LIN {X 9.053,Y 108.159,Z 56.000,A 180.000,B 0.000,C 180.000} C_DIS
LIN {X 9.120,Y 108.308,Z 56.000,A 180.000,B 0.000,C 180.000} C_DIS
LIN {X 9.797,Y 109.768,Z 56.000,A 180.000,B 0.000,C 180.000} C_DIS
LIN {X 9.836,Y 109.849,Z 56.000,A 180.000,B 0.000,C 180.000} C_DIS
LIN {X 10.551,Y 111.303,Z 56.000,A 180.000,B 0.000,C 180.000} C_DIS
LIN {X 10.587,Y 111.377,Z 56.000,A 180.000,B 0.000,C 180.000} C_DIS
LIN {X 10.680,Y 111.556,Z 56.000,A 180.000,B 0.000,C 180.000} C_DIS
LIN {X 11.332,Y 112.807,Z 56.000,A 180.000,B 0.000,C 180.000} C_DIS
LIN {X 11.426,Y 112.986,Z 56.000,A 180.000,B 0.000,C 180.000} C_DIS
LIN {X 12.215,Y 114.416,Z 56.000,A 180.000,B 0.000,C 180.000} C_DIS
LIN {X 12.317,Y 114.595,Z 56.000,A 180.000,B 0.000,C 180.000} C_DIS
LIN {X 13.053,Y 115.859,Z 56.000,A 180.000,B 0.000,C 180.000} C_DIS
LIN {X 13.151,Y 116.025,Z 56.000,A 180.000,B 0.000,C 180.000} C_DIS
LIN {X 13.232,Y 116.158,Z 56.000,A 180.000,B 0.000,C 180.000} C_DIS
LIN {X 14.029,Y 117.455,Z 56.000,A 180.000,B 0.000,C 180.000} C_DIS
LIN {X 14.126,Y 117.607,Z 56.000,A 180.000,B 0.000,C 180.000} C_DIS
LIN {X 14.953,Y 118.885,Z 56.000,A 180.000,B 0.000,C 180.000} C_DIS
LIN {X 15.020,Y 118.988,Z 56.000,A 180.000,B 0.000,C 180.000} C_DIS
LIN {X 15.072,Y 119.064,Z 56.000,A 180.000,B 0.000,C 180.000} C_DIS
LIN {X 15.924,Y 120.315,Z 56.000,A 180.000,B 0.000,C 180.000} C_DIS
LIN {X 16.047,Y 120.494,Z 56.000,A 180.000,B 0.000,C 180.000} C_DIS
LIN {X 16.986,Y 121.806,Z 56.000,A 180.000,B 0.000,C 180.000} C_DIS
LIN {X 17.073,Y 121.924,Z 56.000,A 180.000,B 0.000,C 180.000} C_DIS
LIN {X 18.059,Y 123.235,Z 56.000,A 180.000,B 0.000,C 180.000} C_DIS
LIN {X 18.152,Y 123.354,Z 56.000,A 180.000,B 0.000,C 180.000} C_DIS
LIN {X 19.139,Y 124.606,Z 56.000,A 180.000,B 0.000,C 180.000} C_DIS
LIN {X 19.286,Y 124.785,Z 56.000,A 180.000,B 0.000,C 180.000} C_DIS
LIN {X 20.204,Y 125.894,Z 56.000,A 180.000,B 0.000,C 180.000} C_DIS
LIN {X 20.323,Y 126.036,Z 56.000,A 180.000,B 0.000,C 180.000} C_DIS
LIN {X 21.410,Y 127.287,Z 56.000,A 180.000,B 0.000,C 180.000} C_DIS
LIN {X 21.456,Y 127.340,Z 56.000,A 180.000,B 0.000,C 180.000} C_DIS
LIN {X 21.570,Y 127.466,Z 56.000,A 180.000,B 0.000,C 180.000} C_DIS
LIN {X 22.547,Y 128.539,Z 56.000,A 180.000,B 0.000,C 180.000} C_DIS
LIN {X 22.707,Y 128.711,Z 56.000,A 180.000,B 0.000,C 180.000} C_DIS
LIN {X 23.780,Y 129.835,Z 56.000,A 180.000,B 0.000,C 180.000} C_DIS
LIN {X 23.910,Y 129.969,Z 56.000,A 180.000,B 0.000,C 180.000} C_DIS
LIN {X 25.031,Y 131.090,Z 56.000,A 180.000,B 0.000,C 180.000} C_DIS
LIN {X 25.165,Y 131.220,Z 56.000,A 180.000,B 0.000,C 180.000} C_DIS
LIN {X 26.289,Y 132.293,Z 56.000,A 180.000,B 0.000,C 180.000} C_DIS
LIN {X 26.461,Y 132.453,Z 56.000,A 180.000,B 0.000,C 180.000} C_DIS
LIN {X 27.534,Y 133.430,Z 56.000,A 180.000,B 0.000,C 180.000} C_DIS
LIN {X 27.660,Y 133.544,Z 56.000,A 180.000,B 0.000,C 180.000} C_DIS
LIN {X 27.713,Y 133.590,Z 56.000,A 180.000,B 0.000,C 180.000} C_DIS
LIN {X 28.964,Y 134.677,Z 56.000,A 180.000,B 0.000,C 180.000} C_DIS
LIN {X 29.106,Y 134.796,Z 56.000,A 180.000,B 0.000,C 180.000} C_DIS
LIN {X 30.215,Y 135.714,Z 56.000,A 180.000,B 0.000,C 180.000} C_DIS
LIN {X 30.394,Y 135.861,Z 56.000,A 180.000,B 0.000,C 180.000} C_DIS
LIN {X 31.646,Y 136.848,Z 56.000,A 180.000,B 0.000,C 180.000} C_DIS
LIN {X 31.765,Y 136.941,Z 56.000,A 180.000,B 0.000,C 180.000} C_DIS
LIN {X 33.076,Y 137.927,Z 56.000,A 180.000,B 0.000,C 180.000} C_DIS
LIN {X 33.194,Y 138.014,Z 56.000,A 180.000,B 0.000,C 180.000} C_DIS
LIN {X 34.506,Y 138.953,Z 56.000,A 180.000,B 0.000,C 180.000} C_DIS
LIN {X 34.685,Y 139.076,Z 56.000,A 180.000,B 0.000,C 180.000} C_DIS
LIN {X 35.936,Y 139.928,Z 56.000,A 180.000,B 0.000,C 180.000} C_DIS
LIN {X 36.012,Y 139.980,Z 56.000,A 180.000,B 0.000,C 180.000} C_DIS
LIN {X 36.115,Y 140.047,Z 56.000,A 180.000,B 0.000,C 180.000} C_DIS
LIN {X 37.393,Y 140.874,Z 56.000,A 180.000,B 0.000,C 180.000} C_DIS
LIN {X 37.545,Y 140.971,Z 56.000,A 180.000,B 0.000,C 180.000} C_DIS
LIN {X 38.842,Y 141.768,Z 56.000,A 180.000,B 0.000,C 180.000} C_DIS
LIN {X 38.975,Y 141.849,Z 56.000,A 180.000,B 0.000,C 180.000} C_DIS
LIN {X 39.141,Y 141.947,Z 56.000,A 180.000,B 0.000,C 180.000} C_DIS
LIN {X 40.405,Y 142.683,Z 56.000,A 180.000,B 0.000,C 180.000} C_DIS
LIN {X 40.584,Y 142.785,Z 56.000,A 180.000,B 0.000,C 180.000} C_DIS
LIN {X 42.014,Y 143.574,Z 56.000,A 180.000,B 0.000,C 180.000} C_DIS
LIN {X 42.193,Y 143.668,Z 56.000,A 180.000,B 0.000,C 180.000} C_DIS
LIN {X 43.444,Y 144.320,Z 56.000,A 180.000,B 0.000,C 180.000} C_DIS
LIN {X 43.623,Y 144.413,Z 56.000,A 180.000,B 0.000,C 180.000} C_DIS
LIN {X 43.697,Y 144.449,Z 56.000,A 180.000,B 0.000,C 180.000} C_DIS
LIN {X 45.151,Y 145.164,Z 56.000,A 180.000,B 0.000,C 180.000} C_DIS
LIN {X 45.232,Y 145.203,Z 56.000,A 180.000,B 0.000,C 180.000} C_DIS
LIN {X 46.692,Y 145.880,Z 56.000,A 180.000,B 0.000,C 180.000} C_DIS
LIN {X 46.841,Y 145.947,Z 56.000,A 180.000,B 0.000,C 180.000} C_DIS
LIN {X 48.331,Y 146.595,Z 56.000,A 180.000,B 0.000,C 180.000} C_DIS
LIN {X 48.450,Y 146.645,Z 56.000,A 180.000,B 0.000,C 180.000} C_DIS
LIN {X 49.880,Y 147.227,Z 56.000,A 180.000,B 0.000,C 180.000} C_DIS
LIN {X 50.059,Y 147.299,Z 56.000,A 180.000,B 0.000,C 180.000} C_DIS
LIN {X 51.496,Y 147.846,Z 56.000,A 180.000,B 0.000,C 180.000} C_DIS
LIN {X 51.668,Y 147.911,Z 56.000,A 180.000,B 0.000,C 180.000} C_DIS
LIN {X 51.847,Y 147.974,Z 56.000,A 180.000,B 0.000,C 180.000} C_DIS
LIN {X 52.272,Y 148.125,Z 56.000,A 180.000,B 0.000,C 180.000} C_DIS
; Link Move Starts
LIN {X 52.569,Y 148.230,Z 56.000,A 180.000,B 0.000,C 180.000} C_DIS
LIN {X 52.866,Y 148.335,Z 55.999,A 180.000,B 0.000,C 180.000} C_DIS
LIN {X 53.163,Y 148.440,Z 55.998,A 180.000,B 0.000,C 180.000} C_DIS
LIN {X 53.461,Y 148.542,Z 55.996,A 180.000,B 0.000,C 180.000} C_DIS
LIN {X 53.761,Y 148.640,Z 55.994,A 180.000,B 0.000,C 180.000} C_DIS
LIN {X 54.060,Y 148.738,Z 55.991,A 180.000,B 0.000,C 180.000} C_DIS
LIN {X 54.359,Y 148.836,Z 55.988,A 180.000,B 0.000,C 180.000} C_DIS
LIN {X 54.659,Y 148.934,Z 55.985,A 180.000,B 0.000,C 180.000} C_DIS
LIN {X 54.958,Y 149.032,Z 55.981,A 180.000,B 0.000,C 180.000} C_DIS
LIN {X 55.260,Y 149.124,Z 55.977,A 180.000,B 0.000,C 180.000} C_DIS
LIN {X 55.561,Y 149.215,Z 55.972,A 180.000,B 0.000,C 180.000} C_DIS
LIN {X 55.712,Y 149.260,Z 55.969,A 180.000,B 0.000,C 180.000} C_DIS
LIN {X 55.863,Y 149.306,Z 55.967,A 180.000,B 0.000,C 180.000} C_DIS
LIN {X 56.013,Y 149.351,Z 55.964,A 180.000,B 0.000,C 180.000} C_DIS
LIN {X 56.164,Y 149.397,Z 55.961,A 180.000,B 0.000,C 180.000} C_DIS
LIN {X 56.315,Y 149.442,Z 55.959,A 180.000,B 0.000,C 180.000} C_DIS
LIN {X 56.466,Y 149.488,Z 55.956,A 180.000,B 0.000,C 180.000} C_DIS
LIN {X 56.617,Y 149.533,Z 55.952,A 180.000,B 0.000,C 180.000} C_DIS
LIN {X 56.768,Y 149.577,Z 55.949,A 180.000,B 0.000,C 180.000} C_DIS
LIN {X 56.920,Y 149.619,Z 55.946,A 180.000,B 0.000,C 180.000} C_DIS
LIN {X 57.072,Y 149.661,Z 55.943,A 180.000,B 0.000,C 180.000} C_DIS
LIN {X 57.223,Y 149.703,Z 55.939,A 180.000,B 0.000,C 180.000} C_DIS
LIN {X 57.375,Y 149.745,Z 55.936,A 180.000,B 0.000,C 180.000} C_DIS
LIN {X 57.527,Y 149.786,Z 55.932,A 180.000,B 0.000,C 180.000} C_DIS
LIN {X 57.679,Y 149.828,Z 55.928,A 180.000,B 0.000,C 180.000} C_DIS
LIN {X 57.831,Y 149.870,Z 55.925,A 180.000,B 0.000,C 180.000} C_DIS
LIN {X 57.982,Y 149.912,Z 55.921,A 180.000,B 0.000,C 180.000} C_DIS
LIN {X 58.134,Y 149.954,Z 55.917,A 180.000,B 0.000,C 180.000} C_DIS
LIN {X 58.286,Y 149.996,Z 55.913,A 180.000,B 0.000,C 180.000} C_DIS
LIN {X 58.438,Y 150.037,Z 55.909,A 180.000,B 0.000,C 180.000} C_DIS
LIN {X 58.591,Y 150.075,Z 55.905,A 180.000,B 0.000,C 180.000} C_DIS
LIN {X 58.744,Y 150.113,Z 55.900,A 180.000,B 0.000,C 180.000} C_DIS
LIN {X 58.897,Y 150.152,Z 55.896,A 180.000,B 0.000,C 180.000} C_DIS
LIN {X 59.049,Y 150.190,Z 55.892,A 180.000,B 0.000,C 180.000} C_DIS
LIN {X 59.202,Y 150.229,Z 55.887,A 180.000,B 0.000,C 180.000} C_DIS
LIN {X 59.355,Y 150.267,Z 55.883,A 180.000,B 0.000,C 180.000} C_DIS
LIN {X 59.508,Y 150.305,Z 55.878,A 180.000,B 0.000,C 180.000} C_DIS
LIN {X 59.660,Y 150.344,Z 55.873,A 180.000,B 0.000,C 180.000} C_DIS
LIN {X 59.813,Y 150.382,Z 55.869,A 180.000,B 0.000,C 180.000} C_DIS
LIN {X 59.966,Y 150.420,Z 55.864,A 180.000,B 0.000,C 180.000} C_DIS
LIN {X 60.119,Y 150.458,Z 55.859,A 180.000,B 0.000,C 180.000} C_DIS
LIN {X 60.272,Y 150.493,Z 55.854,A 180.000,B 0.000,C 180.000} C_DIS
LIN {X 60.349,Y 150.510,Z 55.851,A 180.000,B 0.000,C 180.000} C_DIS
LIN {X 60.426,Y 150.527,Z 55.849,A 180.000,B 0.000,C 180.000} C_DIS
LIN {X 60.503,Y 150.545,Z 55.846,A 180.000,B 0.000,C 180.000} C_DIS
LIN {X 60.580,Y 150.562,Z 55.844,A 180.000,B 0.000,C 180.000} C_DIS
LIN {X 60.656,Y 150.580,Z 55.841,A 180.000,B 0.000,C 180.000} C_DIS
LIN {X 60.733,Y 150.597,Z 55.839,A 180.000,B 0.000,C 180.000} C_DIS
LIN {X 60.810,Y 150.614,Z 55.836,A 180.000,B 0.000,C 180.000} C_DIS
LIN {X 60.964,Y 150.649,Z 55.831,A 180.000,B 0.000,C 180.000} C_DIS
LIN {X 61.117,Y 150.684,Z 55.825,A 180.000,B 0.000,C 180.000} C_DIS
LIN {X 61.271,Y 150.719,Z 55.820,A 180.000,B 0.000,C 180.000} C_DIS
LIN {X 61.424,Y 150.754,Z 55.815,A 180.000,B 0.000,C 180.000} C_DIS
LIN {X 61.578,Y 150.788,Z 55.809,A 180.000,B 0.000,C 180.000} C_DIS
LIN {X 61.655,Y 150.806,Z 55.806,A 180.000,B 0.000,C 180.000} C_DIS
LIN {X 61.732,Y 150.823,Z 55.804,A 180.000,B 0.000,C 180.000} C_DIS
LIN {X 61.809,Y 150.840,Z 55.801,A 180.000,B 0.000,C 180.000} C_DIS
LIN {X 61.886,Y 150.856,Z 55.798,A 180.000,B 0.000,C 180.000} C_DIS
LIN {X 61.963,Y 150.871,Z 55.796,A 180.000,B 0.000,C 180.000} C_DIS
LIN {X 62.117,Y 150.902,Z 55.790,A 180.000,B 0.000,C 180.000} C_DIS
LIN {X 62.349,Y 150.949,Z 55.782,A 180.000,B 0.000,C 180.000} C_DIS
LIN {X 62.503,Y 150.980,Z 55.776,A 180.000,B 0.000,C 180.000} C_DIS
LIN {X 62.581,Y 150.996,Z 55.774,A 180.000,B 0.000,C 180.000} C_DIS
LIN {X 62.735,Y 151.027,Z 55.768,A 180.000,B 0.000,C 180.000} C_DIS
LIN {X 62.966,Y 151.074,Z 55.760,A 180.000,B 0.000,C 180.000} C_DIS
LIN {X 63.121,Y 151.105,Z 55.754,A 180.000,B 0.000,C 180.000} C_DIS
LIN {X 63.198,Y 151.121,Z 55.752,A 180.000,B 0.000,C 180.000} C_DIS
LIN {X 63.352,Y 151.152,Z 55.746,A 180.000,B 0.000,C 180.000} C_DIS
LIN {X 63.430,Y 151.168,Z 55.743,A 180.000,B 0.000,C 180.000} C_DIS
LIN {X 63.507,Y 151.183,Z 55.741,A 180.000,B 0.000,C 180.000} C_DIS
LIN {X 63.584,Y 151.197,Z 55.738,A 180.000,B 0.000,C 180.000} C_DIS
LIN {X 63.739,Y 151.225,Z 55.732,A 180.000,B 0.000,C 180.000} C_DIS
LIN {X 63.817,Y 151.238,Z 55.730,A 180.000,B 0.000,C 180.000} C_DIS
LIN {X 63.972,Y 151.266,Z 55.724,A 180.000,B 0.000,C 180.000} C_DIS
LIN {X 64.437,Y 151.349,Z 55.708,A 180.000,B 0.000,C 180.000} C_DIS
LIN {X 64.592,Y 151.376,Z 55.702,A 180.000,B 0.000,C 180.000} C_DIS
LIN {X 65.057,Y 151.459,Z 55.686,A 180.000,B 0.000,C 180.000} C_DIS
LIN {X 65.213,Y 151.486,Z 55.680,A 180.000,B 0.000,C 180.000} C_DIS
LIN {X 65.290,Y 151.499,Z 55.677,A 180.000,B 0.000,C 180.000} C_DIS
LIN {X 65.368,Y 151.511,Z 55.675,A 180.000,B 0.000,C 180.000} C_DIS
LIN {X 65.524,Y 151.535,Z 55.669,A 180.000,B 0.000,C 180.000} C_DIS
LIN {X 66.069,Y 151.619,Z 55.650,A 180.000,B 0.000,C 180.000} C_DIS
LIN {X 66.536,Y 151.690,Z 55.633,A 180.000,B 0.000,C 180.000} C_DIS
LIN {X 66.691,Y 151.714,Z 55.628,A 180.000,B 0.000,C 180.000} C_DIS
LIN {X 66.925,Y 151.750,Z 55.620,A 180.000,B 0.000,C 180.000} C_DIS
LIN {X 67.003,Y 151.762,Z 55.617,A 180.000,B 0.000,C 180.000} C_DIS
LIN {X 67.081,Y 151.772,Z 55.614,A 180.000,B 0.000,C 180.000} C_DIS
LIN {X 67.862,Y 151.873,Z 55.587,A 180.000,B 0.000,C 180.000} C_DIS
LIN {X 68.252,Y 151.924,Z 55.573,A 180.000,B 0.000,C 180.000} C_DIS
LIN {X 68.643,Y 151.974,Z 55.559,A 180.000,B 0.000,C 180.000} C_DIS
LIN {X 68.721,Y 151.984,Z 55.556,A 180.000,B 0.000,C 180.000} C_DIS
LIN {X 68.799,Y 151.993,Z 55.554,A 180.000,B 0.000,C 180.000} C_DIS
LIN {X 69.347,Y 152.051,Z 55.534,A 180.000,B 0.000,C 180.000} C_DIS
LIN {X 70.130,Y 152.134,Z 55.507,A 180.000,B 0.000,C 180.000} C_DIS
LIN {X 70.444,Y 152.167,Z 55.496,A 180.000,B 0.000,C 180.000} C_DIS
LIN {X 70.522,Y 152.174,Z 55.493,A 180.000,B 0.000,C 180.000} C_DIS
LIN {X 72.170,Y 152.310,Z 55.435,A 180.000,B 0.000,C 180.000} C_DIS
LIN {X 72.249,Y 152.316,Z 55.433,A 180.000,B 0.000,C 180.000} C_DIS
LIN {X 72.327,Y 152.321,Z 55.430,A 180.000,B 0.000,C 180.000} C_DIS
LIN {X 73.428,Y 152.385,Z 55.391,A 180.000,B 0.000,C 180.000} C_DIS
LIN {X 73.585,Y 152.394,Z 55.386,A 180.000,B 0.000,C 180.000} C_DIS
LIN {X 73.900,Y 152.413,Z 55.375,A 180.000,B 0.000,C 180.000} C_DIS
LIN {X 73.978,Y 152.417,Z 55.372,A 180.000,B 0.000,C 180.000} C_DIS
LIN {X 74.057,Y 152.420,Z 55.369,A 180.000,B 0.000,C 180.000} C_DIS
LIN {X 74.214,Y 152.426,Z 55.364,A 180.000,B 0.000,C 180.000} C_DIS
LIN {X 74.687,Y 152.442,Z 55.347,A 180.000,B 0.000,C 180.000} C_DIS
LIN {X 74.844,Y 152.448,Z 55.342,A 180.000,B 0.000,C 180.000} C_DIS
LIN {X 75.316,Y 152.465,Z 55.325,A 180.000,B 0.000,C 180.000} C_DIS
LIN {X 75.395,Y 152.467,Z 55.323,A 180.000,B 0.000,C 180.000} C_DIS
LIN {X 75.552,Y 152.473,Z 55.317,A 180.000,B 0.000,C 180.000} C_DIS
LIN {X 75.710,Y 152.478,Z 55.312,A 180.000,B 0.000,C 180.000} C_DIS
LIN {X 75.789,Y 152.480,Z 55.309,A 180.000,B 0.000,C 180.000} C_DIS
LIN {X 75.946,Y 152.482,Z 55.303,A 180.000,B 0.000,C 180.000} C_DIS
LIN {X 76.025,Y 152.483,Z 55.301,A 180.000,B 0.000,C 180.000} C_DIS
LIN {X 76.182,Y 152.485,Z 55.295,A 180.000,B 0.000,C 180.000} C_DIS
LIN {X 76.655,Y 152.490,Z 55.279,A 180.000,B 0.000,C 180.000} C_DIS
LIN {X 76.812,Y 152.492,Z 55.273,A 180.000,B 0.000,C 180.000} C_DIS
LIN {X 77.048,Y 152.495,Z 55.265,A 180.000,B 0.000,C 180.000} C_DIS
LIN {X 77.206,Y 152.497,Z 55.259,A 180.000,B 0.000,C 180.000} C_DIS
LIN {X 77.285,Y 152.498,Z 55.257,A 180.000,B 0.000,C 180.000} C_DIS
LIN {X 77.442,Y 152.499,Z 55.251,A 180.000,B 0.000,C 180.000} C_DIS
LIN {X 77.521,Y 152.500,Z 55.248,A 180.000,B 0.000,C 180.000} C_DIS
LIN {X 77.600,Y 152.499,Z 55.246,A 180.000,B 0.000,C 180.000} C_DIS
LIN {X 77.757,Y 152.497,Z 55.240,A 180.000,B 0.000,C 180.000} C_DIS
LIN {X 77.993,Y 152.494,Z 55.232,A 180.000,B 0.000,C 180.000} C_DIS
LIN {X 78.151,Y 152.493,Z 55.226,A 180.000,B 0.000,C 180.000} C_DIS
LIN {X 78.230,Y 152.492,Z 55.224,A 180.000,B 0.000,C 180.000} C_DIS
LIN {X 78.387,Y 152.490,Z 55.218,A 180.000,B 0.000,C 180.000} C_DIS
LIN {X 78.623,Y 152.487,Z 55.210,A 180.000,B 0.000,C 180.000} C_DIS
LIN {X 78.781,Y 152.485,Z 55.204,A 180.000,B 0.000,C 180.000} C_DIS
LIN {X 78.860,Y 152.484,Z 55.202,A 180.000,B 0.000,C 180.000} C_DIS
LIN {X 79.017,Y 152.482,Z 55.196,A 180.000,B 0.000,C 180.000} C_DIS
LIN {X 79.175,Y 152.481,Z 55.191,A 180.000,B 0.000,C 180.000} C_DIS
LIN {X 79.253,Y 152.479,Z 55.188,A 180.000,B 0.000,C 180.000} C_DIS
LIN {X 79.332,Y 152.477,Z 55.185,A 180.000,B 0.000,C 180.000} C_DIS
LIN {X 79.489,Y 152.471,Z 55.180,A 180.000,B 0.000,C 180.000} C_DIS
LIN {X 79.647,Y 152.466,Z 55.174,A 180.000,B 0.000,C 180.000} C_DIS
LIN {X 79.804,Y 152.460,Z 55.169,A 180.000,B 0.000,C 180.000} C_DIS
LIN {X 79.962,Y 152.455,Z 55.164,A 180.000,B 0.000,C 180.000} C_DIS
LIN {X 80.040,Y 152.452,Z 55.161,A 180.000,B 0.000,C 180.000} C_DIS
LIN {X 80.119,Y 152.449,Z 55.159,A 180.000,B 0.000,C 180.000} C_DIS
LIN {X 80.198,Y 152.447,Z 55.156,A 180.000,B 0.000,C 180.000} C_DIS
LIN {X 80.276,Y 152.444,Z 55.154,A 180.000,B 0.000,C 180.000} C_DIS
LIN {X 80.355,Y 152.441,Z 55.151,A 180.000,B 0.000,C 180.000} C_DIS
LIN {X 80.434,Y 152.438,Z 55.148,A 180.000,B 0.000,C 180.000} C_DIS
LIN {X 80.591,Y 152.433,Z 55.143,A 180.000,B 0.000,C 180.000} C_DIS
LIN {X 80.749,Y 152.427,Z 55.139,A 180.000,B 0.000,C 180.000} C_DIS
LIN {X 80.906,Y 152.422,Z 55.134,A 180.000,B 0.000,C 180.000} C_DIS
LIN {X 81.063,Y 152.415,Z 55.129,A 180.000,B 0.000,C 180.000} C_DIS
LIN {X 81.221,Y 152.406,Z 55.124,A 180.000,B 0.000,C 180.000} C_DIS
LIN {X 81.378,Y 152.396,Z 55.120,A 180.000,B 0.000,C 180.000} C_DIS
LIN {X 81.535,Y 152.387,Z 55.115,A 180.000,B 0.000,C 180.000} C_DIS
LIN {X 81.692,Y 152.378,Z 55.110,A 180.000,B 0.000,C 180.000} C_DIS
LIN {X 81.850,Y 152.369,Z 55.106,A 180.000,B 0.000,C 180.000} C_DIS
LIN {X 82.007,Y 152.360,Z 55.102,A 180.000,B 0.000,C 180.000} C_DIS
LIN {X 82.164,Y 152.350,Z 55.097,A 180.000,B 0.000,C 180.000} C_DIS
LIN {X 82.321,Y 152.341,Z 55.093,A 180.000,B 0.000,C 180.000} C_DIS
LIN {X 82.478,Y 152.332,Z 55.089,A 180.000,B 0.000,C 180.000} C_DIS
LIN {X 82.636,Y 152.323,Z 55.085,A 180.000,B 0.000,C 180.000} C_DIS
LIN {X 82.793,Y 152.313,Z 55.081,A 180.000,B 0.000,C 180.000} C_DIS
LIN {X 82.950,Y 152.300,Z 55.077,A 180.000,B 0.000,C 180.000} C_DIS
LIN {X 83.107,Y 152.287,Z 55.073,A 180.000,B 0.000,C 180.000} C_DIS
LIN {X 83.264,Y 152.274,Z 55.070,A 180.000,B 0.000,C 180.000} C_DIS
LIN {X 83.421,Y 152.261,Z 55.066,A 180.000,B 0.000,C 180.000} C_DIS
LIN {X 83.578,Y 152.248,Z 55.062,A 180.000,B 0.000,C 180.000} C_DIS
LIN {X 83.735,Y 152.235,Z 55.059,A 180.000,B 0.000,C 180.000} C_DIS
LIN {X 83.892,Y 152.223,Z 55.056,A 180.000,B 0.000,C 180.000} C_DIS
LIN {X 84.049,Y 152.210,Z 55.052,A 180.000,B 0.000,C 180.000} C_DIS
LIN {X 84.206,Y 152.197,Z 55.049,A 180.000,B 0.000,C 180.000} C_DIS
LIN {X 84.363,Y 152.184,Z 55.046,A 180.000,B 0.000,C 180.000} C_DIS
LIN {X 84.520,Y 152.171,Z 55.043,A 180.000,B 0.000,C 180.000} C_DIS
LIN {X 84.676,Y 152.154,Z 55.040,A 180.000,B 0.000,C 180.000} C_DIS
LIN {X 84.833,Y 152.138,Z 55.037,A 180.000,B 0.000,C 180.000} C_DIS
LIN {X 84.989,Y 152.121,Z 55.034,A 180.000,B 0.000,C 180.000} C_DIS
LIN {X 85.146,Y 152.105,Z 55.032,A 180.000,B 0.000,C 180.000} C_DIS
LIN {X 85.303,Y 152.088,Z 55.029,A 180.000,B 0.000,C 180.000} C_DIS
LIN {X 85.459,Y 152.071,Z 55.027,A 180.000,B 0.000,C 180.000} C_DIS
LIN {X 85.773,Y 152.038,Z 55.022,A 180.000,B 0.000,C 180.000} C_DIS
LIN {X 86.086,Y 152.005,Z 55.018,A 180.000,B 0.000,C 180.000} C_DIS
LIN {X 86.399,Y 151.969,Z 55.014,A 180.000,B 0.000,C 180.000} C_DIS
LIN {X 86.711,Y 151.928,Z 55.011,A 180.000,B 0.000,C 180.000} C_DIS
LIN {X 87.023,Y 151.888,Z 55.008,A 180.000,B 0.000,C 180.000} C_DIS
LIN {X 87.336,Y 151.847,Z 55.005,A 180.000,B 0.000,C 180.000} C_DIS
LIN {X 87.648,Y 151.807,Z 55.003,A 180.000,B 0.000,C 180.000} C_DIS
LIN {X 87.961,Y 151.766,Z 55.002,A 180.000,B 0.000,C 180.000} C_DIS
LIN {X 88.272,Y 151.720,Z 55.001,A 180.000,B 0.000,C 180.000} C_DIS
LIN {X 88.583,Y 151.672,Z 55.000,A 180.000,B 0.000,C 180.000} C_DIS
LIN {X 88.812,Y 151.637,Z 55.000,A 180.000,B 0.000,C 180.000} C_DIS
; Cutting Move Starts
LIN {X 89.567,Y 151.521,Z 55.000,A 180.000,B 0.000,C 180.000} C_DIS
LIN {X 89.746,Y 151.494,Z 55.000,A 180.000,B 0.000,C 180.000} C_DIS
LIN {X 89.925,Y 151.462,Z 55.000,A 180.000,B 0.000,C 180.000} C_DIS
LIN {X 91.355,Y 151.208,Z 55.000,A 180.000,B 0.000,C 180.000} C_DIS
LIN {X 91.533,Y 151.175,Z 55.000,A 180.000,B 0.000,C 180.000} C_DIS
LIN {X 93.142,Y 150.850,Z 55.000,A 180.000,B 0.000,C 180.000} C_DIS
LIN {X 93.321,Y 150.811,Z 55.000,A 180.000,B 0.000,C 180.000} C_DIS
LIN {X 94.751,Y 150.487,Z 55.000,A 180.000,B 0.000,C 180.000} C_DIS
LIN {X 94.930,Y 150.447,Z 55.000,A 180.000,B 0.000,C 180.000} C_DIS
LIN {X 95.109,Y 150.402,Z 55.000,A 180.000,B 0.000,C 180.000} C_DIS
LIN {X 96.539,Y 150.042,Z 55.000,A 180.000,B 0.000,C 180.000} C_DIS
LIN {X 96.718,Y 149.995,Z 55.000,A 180.000,B 0.000,C 180.000} C_DIS
LIN {X 98.148,Y 149.600,Z 55.000,A 180.000,B 0.000,C 180.000} C_DIS
LIN {X 98.327,Y 149.550,Z 55.000,A 180.000,B 0.000,C 180.000} C_DIS
LIN {X 98.505,Y 149.497,Z 55.000,A 180.000,B 0.000,C 180.000} C_DIS
LIN {X 99.936,Y 149.065,Z 55.000,A 180.000,B 0.000,C 180.000} C_DIS
LIN {X 100.114,Y 149.008,Z 55.000,A 180.000,B 0.000,C 180.000} C_DIS
LIN {X 101.545,Y 148.540,Z 55.000,A 180.000,B 0.000,C 180.000} C_DIS
LIN {X 101.723,Y 148.480,Z 55.000,A 180.000,B 0.000,C 180.000} C_DIS
LIN {X 103.153,Y 147.974,Z 55.000,A 180.000,B 0.000,C 180.000} C_DIS
LIN {X 103.332,Y 147.911,Z 55.000,A 180.000,B 0.000,C 180.000} C_DIS
LIN {X 103.504,Y 147.846,Z 55.000,A 180.000,B 0.000,C 180.000} C_DIS
LIN {X 104.941,Y 147.299,Z 55.000,A 180.000,B 0.000,C 180.000} C_DIS
LIN {X 105.120,Y 147.227,Z 55.000,A 180.000,B 0.000,C 180.000} C_DIS
LIN {X 106.550,Y 146.645,Z 55.000,A 180.000,B 0.000,C 180.000} C_DIS
LIN {X 106.669,Y 146.595,Z 55.000,A 180.000,B 0.000,C 180.000} C_DIS
LIN {X 108.159,Y 145.947,Z 55.000,A 180.000,B 0.000,C 180.000} C_DIS
LIN {X 108.308,Y 145.880,Z 55.000,A 180.000,B 0.000,C 180.000} C_DIS
LIN {X 109.768,Y 145.203,Z 55.000,A 180.000,B 0.000,C 180.000} C_DIS
LIN {X 109.849,Y 145.164,Z 55.000,A 180.000,B 0.000,C 180.000} C_DIS
LIN {X 111.303,Y 144.449,Z 55.000,A 180.000,B 0.000,C 180.000} C_DIS
LIN {X 111.377,Y 144.413,Z 55.000,A 180.000,B 0.000,C 180.000} C_DIS
LIN {X 111.556,Y 144.320,Z 55.000,A 180.000,B 0.000,C 180.000} C_DIS
LIN {X 112.807,Y 143.668,Z 55.000,A 180.000,B 0.000,C 180.000} C_DIS
LIN {X 112.986,Y 143.574,Z 55.000,A 180.000,B 0.000,C 180.000} C_DIS
LIN {X 114.416,Y 142.785,Z 55.000,A 180.000,B 0.000,C 180.000} C_DIS
LIN {X 114.595,Y 142.683,Z 55.000,A 180.000,B 0.000,C 180.000} C_DIS
LIN {X 115.859,Y 141.947,Z 55.000,A 180.000,B 0.000,C 180.000} C_DIS
LIN {X 116.025,Y 141.849,Z 55.000,A 180.000,B 0.000,C 180.000} C_DIS
LIN {X 116.158,Y 141.768,Z 55.000,A 180.000,B 0.000,C 180.000} C_DIS
LIN {X 117.455,Y 140.971,Z 55.000,A 180.000,B 0.000,C 180.000} C_DIS
LIN {X 117.607,Y 140.874,Z 55.000,A 180.000,B 0.000,C 180.000} C_DIS
LIN {X 118.885,Y 140.047,Z 55.000,A 180.000,B 0.000,C 180.000} C_DIS
LIN {X 118.988,Y 139.980,Z 55.000,A 180.000,B 0.000,C 180.000} C_DIS
LIN {X 119.064,Y 139.928,Z 55.000,A 180.000,B 0.000,C 180.000} C_DIS
LIN {X 120.315,Y 139.076,Z 55.000,A 180.000,B 0.000,C 180.000} C_DIS
LIN {X 120.494,Y 138.953,Z 55.000,A 180.000,B 0.000,C 180.000} C_DIS
LIN {X 121.806,Y 138.014,Z 55.000,A 180.000,B 0.000,C 180.000} C_DIS
LIN {X 121.924,Y 137.927,Z 55.000,A 180.000,B 0.000,C 180.000} C_DIS
LIN {X 123.235,Y 136.941,Z 55.000,A 180.000,B 0.000,C 180.000} C_DIS
LIN {X 123.354,Y 136.848,Z 55.000,A 180.000,B 0.000,C 180.000} C_DIS
LIN {X 124.606,Y 135.861,Z 55.000,A 180.000,B 0.000,C 180.000} C_DIS
LIN {X 124.785,Y 135.714,Z 55.000,A 180.000,B 0.000,C 180.000} C_DIS
LIN {X 125.894,Y 134.796,Z 55.000,A 180.000,B 0.000,C 180.000} C_DIS
LIN {X 126.036,Y 134.677,Z 55.000,A 180.000,B 0.000,C 180.000} C_DIS
LIN {X 127.287,Y 133.590,Z 55.000,A 180.000,B 0.000,C 180.000} C_DIS
LIN {X 127.340,Y 133.544,Z 55.000,A 180.000,B 0.000,C 180.000} C_DIS
LIN {X 127.466,Y 133.430,Z 55.000,A 180.000,B 0.000,C 180.000} C_DIS
LIN {X 128.539,Y 132.453,Z 55.000,A 180.000,B 0.000,C 180.000} C_DIS
LIN {X 128.711,Y 132.293,Z 55.000,A 180.000,B 0.000,C 180.000} C_DIS
LIN {X 129.835,Y 131.220,Z 55.000,A 180.000,B 0.000,C 180.000} C_DIS
LIN {X 129.969,Y 131.090,Z 55.000,A 180.000,B 0.000,C 180.000} C_DIS
LIN {X 131.090,Y 129.969,Z 55.000,A 180.000,B 0.000,C 180.000} C_DIS
LIN {X 131.220,Y 129.835,Z 55.000,A 180.000,B 0.000,C 180.000} C_DIS
LIN {X 132.293,Y 128.711,Z 55.000,A 180.000,B 0.000,C 180.000} C_DIS
LIN {X 132.453,Y 128.539,Z 55.000,A 180.000,B 0.000,C 180.000} C_DIS
LIN {X 133.430,Y 127.466,Z 55.000,A 180.000,B 0.000,C 180.000} C_DIS
LIN {X 133.544,Y 127.340,Z 55.000,A 180.000,B 0.000,C 180.000} C_DIS
LIN {X 133.590,Y 127.287,Z 55.000,A 180.000,B 0.000,C 180.000} C_DIS
LIN {X 134.677,Y 126.036,Z 55.000,A 180.000,B 0.000,C 180.000} C_DIS
LIN {X 134.796,Y 125.894,Z 55.000,A 180.000,B 0.000,C 180.000} C_DIS
LIN {X 135.714,Y 124.785,Z 55.000,A 180.000,B 0.000,C 180.000} C_DIS
LIN {X 135.861,Y 124.606,Z 55.000,A 180.000,B 0.000,C 180.000} C_DIS
LIN {X 136.848,Y 123.354,Z 55.000,A 180.000,B 0.000,C 180.000} C_DIS
LIN {X 136.941,Y 123.235,Z 55.000,A 180.000,B 0.000,C 180.000} C_DIS
LIN {X 137.927,Y 121.924,Z 55.000,A 180.000,B 0.000,C 180.000} C_DIS
LIN {X 138.014,Y 121.806,Z 55.000,A 180.000,B 0.000,C 180.000} C_DIS
LIN {X 138.953,Y 120.494,Z 55.000,A 180.000,B 0.000,C 180.000} C_DIS
LIN {X 139.076,Y 120.315,Z 55.000,A 180.000,B 0.000,C 180.000} C_DIS
LIN {X 139.928,Y 119.064,Z 55.000,A 180.000,B 0.000,C 180.000} C_DIS
LIN {X 139.980,Y 118.988,Z 55.000,A 180.000,B 0.000,C 180.000} C_DIS
LIN {X 140.047,Y 118.885,Z 55.000,A 180.000,B 0.000,C 180.000} C_DIS
LIN {X 140.874,Y 117.607,Z 55.000,A 180.000,B 0.000,C 180.000} C_DIS
LIN {X 140.971,Y 117.455,Z 55.000,A 180.000,B 0.000,C 180.000} C_DIS
LIN {X 141.768,Y 116.158,Z 55.000,A 180.000,B 0.000,C 180.000} C_DIS
LIN {X 141.849,Y 116.025,Z 55.000,A 180.000,B 0.000,C 180.000} C_DIS
LIN {X 141.947,Y 115.859,Z 55.000,A 180.000,B 0.000,C 180.000} C_DIS
LIN {X 142.683,Y 114.595,Z 55.000,A 180.000,B 0.000,C 180.000} C_DIS
LIN {X 142.785,Y 114.416,Z 55.000,A 180.000,B 0.000,C 180.000} C_DIS
LIN {X 143.574,Y 112.986,Z 55.000,A 180.000,B 0.000,C 180.000} C_DIS
LIN {X 143.668,Y 112.807,Z 55.000,A 180.000,B 0.000,C 180.000} C_DIS
LIN {X 144.320,Y 111.556,Z 55.000,A 180.000,B 0.000,C 180.000} C_DIS
LIN {X 144.413,Y 111.377,Z 55.000,A 180.000,B 0.000,C 180.000} C_DIS
LIN {X 144.449,Y 111.303,Z 55.000,A 180.000,B 0.000,C 180.000} C_DIS
LIN {X 145.164,Y 109.849,Z 55.000,A 180.000,B 0.000,C 180.000} C_DIS
LIN {X 145.203,Y 109.768,Z 55.000,A 180.000,B 0.000,C 180.000} C_DIS
LIN {X 145.880,Y 108.308,Z 55.000,A 180.000,B 0.000,C 180.000} C_DIS
LIN {X 145.947,Y 108.159,Z 55.000,A 180.000,B 0.000,C 180.000} C_DIS
LIN {X 146.595,Y 106.669,Z 55.000,A 180.000,B 0.000,C 180.000} C_DIS
LIN {X 146.645,Y 106.550,Z 55.000,A 180.000,B 0.000,C 180.000} C_DIS
LIN {X 147.227,Y 105.120,Z 55.000,A 180.000,B 0.000,C 180.000} C_DIS
LIN {X 147.299,Y 104.941,Z 55.000,A 180.000,B 0.000,C 180.000} C_DIS
LIN {X 147.846,Y 103.504,Z 55.000,A 180.000,B 0.000,C 180.000} C_DIS
LIN {X 147.911,Y 103.332,Z 55.000,A 180.000,B 0.000,C 180.000} C_DIS
LIN {X 147.974,Y 103.153,Z 55.000,A 180.000,B 0.000,C 180.000} C_DIS
LIN {X 148.480,Y 101.723,Z 55.000,A 180.000,B 0.000,C 180.000} C_DIS
LIN {X 148.540,Y 101.545,Z 55.000,A 180.000,B 0.000,C 180.000} C_DIS
LIN {X 149.008,Y 100.114,Z 55.000,A 180.000,B 0.000,C 180.000} C_DIS
LIN {X 149.065,Y 99.936,Z 55.000,A 180.000,B 0.000,C 180.000} C_DIS
LIN {X 149.497,Y 98.505,Z 55.000,A 180.000,B 0.000,C 180.000} C_DIS
LIN {X 149.550,Y 98.327,Z 55.000,A 180.000,B 0.000,C 180.000} C_DIS
LIN {X 149.600,Y 98.148,Z 55.000,A 180.000,B 0.000,C 180.000} C_DIS
LIN {X 149.995,Y 96.718,Z 55.000,A 180.000,B 0.000,C 180.000} C_DIS
LIN {X 150.042,Y 96.539,Z 55.000,A 180.000,B 0.000,C 180.000} C_DIS
LIN {X 150.402,Y 95.109,Z 55.000,A 180.000,B 0.000,C 180.000} C_DIS
LIN {X 150.447,Y 94.930,Z 55.000,A 180.000,B 0.000,C 180.000} C_DIS
LIN {X 150.487,Y 94.751,Z 55.000,A 180.000,B 0.000,C 180.000} C_DIS
LIN {X 150.811,Y 93.321,Z 55.000,A 180.000,B 0.000,C 180.000} C_DIS
LIN {X 150.850,Y 93.142,Z 55.000,A 180.000,B 0.000,C 180.000} C_DIS
LIN {X 151.175,Y 91.533,Z 55.000,A 180.000,B 0.000,C 180.000} C_DIS
LIN {X 151.208,Y 91.355,Z 55.000,A 180.000,B 0.000,C 180.000} C_DIS
LIN {X 151.462,Y 89.925,Z 55.000,A 180.000,B 0.000,C 180.000} C_DIS
LIN {X 151.494,Y 89.746,Z 55.000,A 180.000,B 0.000,C 180.000} C_DIS
LIN {X 151.521,Y 89.567,Z 55.000,A 180.000,B 0.000,C 180.000} C_DIS
LIN {X 151.741,Y 88.137,Z 55.000,A 180.000,B 0.000,C 180.000} C_DIS
LIN {X 151.767,Y 87.958,Z 55.000,A 180.000,B 0.000,C 180.000} C_DIS
LIN {X 151.975,Y 86.349,Z 55.000,A 180.000,B 0.000,C 180.000} C_DIS
LIN {X 151.996,Y 86.170,Z 55.000,A 180.000,B 0.000,C 180.000} C_DIS
LIN {X 152.167,Y 84.561,Z 55.000,A 180.000,B 0.000,C 180.000} C_DIS
LIN {X 152.182,Y 84.383,Z 55.000,A 180.000,B 0.000,C 180.000} C_DIS
LIN {X 152.300,Y 82.952,Z 55.000,A 180.000,B 0.000,C 180.000} C_DIS
LIN {X 152.314,Y 82.774,Z 55.000,A 180.000,B 0.000,C 180.000} C_DIS
LIN {X 152.315,Y 82.761,Z 55.000,A 180.000,B 0.000,C 180.000} C_DIS
LIN {X 152.325,Y 82.595,Z 55.000,A 180.000,B 0.000,C 180.000} C_DIS
LIN {X 152.409,Y 81.165,Z 55.000,A 180.000,B 0.000,C 180.000} C_DIS
LIN {X 152.419,Y 80.986,Z 55.000,A 180.000,B 0.000,C 180.000} C_DIS
LIN {X 152.475,Y 79.377,Z 55.000,A 180.000,B 0.000,C 180.000} C_DIS
LIN {X 152.480,Y 79.198,Z 55.000,A 180.000,B 0.000,C 180.000} C_DIS
LIN {X 152.499,Y 77.589,Z 55.000,A 180.000,B 0.000,C 180.000} C_DIS
LIN {X 152.499,Y 77.411,Z 55.000,A 180.000,B 0.000,C 180.000} C_DIS
LIN {X 152.480,Y 75.802,Z 55.000,A 180.000,B 0.000,C 180.000} C_DIS
LIN {X 152.475,Y 75.623,Z 55.000,A 180.000,B 0.000,C 180.000} C_DIS
LIN {X 152.419,Y 74.014,Z 55.000,A 180.000,B 0.000,C 180.000} C_DIS
LIN {X 152.409,Y 73.835,Z 55.000,A 180.000,B 0.000,C 180.000} C_DIS
LIN {X 152.325,Y 72.405,Z 55.000,A 180.000,B 0.000,C 180.000} C_DIS
LIN {X 152.315,Y 72.239,Z 55.000,A 180.000,B 0.000,C 180.000} C_DIS
LIN {X 152.314,Y 72.226,Z 55.000,A 180.000,B 0.000,C 180.000} C_DIS
LIN {X 152.300,Y 72.048,Z 55.000,A 180.000,B 0.000,C 180.000} C_DIS
LIN {X 152.182,Y 70.617,Z 55.000,A 180.000,B 0.000,C 180.000} C_DIS
LIN {X 152.167,Y 70.439,Z 55.000,A 180.000,B 0.000,C 180.000} C_DIS
LIN {X 151.996,Y 68.830,Z 55.000,A 180.000,B 0.000,C 180.000} C_DIS
LIN {X 151.975,Y 68.651,Z 55.000,A 180.000,B 0.000,C 180.000} C_DIS
LIN {X 151.767,Y 67.042,Z 55.000,A 180.000,B 0.000,C 180.000} C_DIS
LIN {X 151.741,Y 66.863,Z 55.000,A 180.000,B 0.000,C 180.000} C_DIS
LIN {X 151.521,Y 65.433,Z 55.000,A 180.000,B 0.000,C 180.000} C_DIS
LIN {X 151.494,Y 65.254,Z 55.000,A 180.000,B 0.000,C 180.000} C_DIS
LIN {X 151.462,Y 65.075,Z 55.000,A 180.000,B 0.000,C 180.000} C_DIS
LIN {X 151.208,Y 63.645,Z 55.000,A 180.000,B 0.000,C 180.000} C_DIS
LIN {X 151.175,Y 63.467,Z 55.000,A 180.000,B 0.000,C 180.000} C_DIS
LIN {X 150.850,Y 61.858,Z 55.000,A 180.000,B 0.000,C 180.000} C_DIS
LIN {X 150.811,Y 61.679,Z 55.000,A 180.000,B 0.000,C 180.000} C_DIS
LIN {X 150.487,Y 60.249,Z 55.000,A 180.000,B 0.000,C 180.000} C_DIS
LIN {X 150.447,Y 60.070,Z 55.000,A 180.000,B 0.000,C 180.000} C_DIS
LIN {X 150.402,Y 59.891,Z 55.000,A 180.000,B 0.000,C 180.000} C_DIS
LIN {X 150.042,Y 58.461,Z 55.000,A 180.000,B 0.000,C 180.000} C_DIS
LIN {X 149.995,Y 58.282,Z 55.000,A 180.000,B 0.000,C 180.000} C_DIS
LIN {X 149.600,Y 56.852,Z 55.000,A 180.000,B 0.000,C 180.000} C_DIS
LIN {X 149.550,Y 56.673,Z 55.000,A 180.000,B 0.000,C 180.000} C_DIS
LIN {X 149.497,Y 56.495,Z 55.000,A 180.000,B 0.000,C 180.000} C_DIS
LIN {X 149.065,Y 55.064,Z 55.000,A 180.000,B 0.000,C 180.000} C_DIS
LIN {X 149.008,Y 54.886,Z 55.000,A 180.000,B 0.000,C 180.000} C_DIS
LIN {X 148.540,Y 53.455,Z 55.000,A 180.000,B 0.000,C 180.000} C_DIS
LIN {X 148.480,Y 53.277,Z 55.000,A 180.000,B 0.000,C 180.000} C_DIS
LIN {X 147.974,Y 51.847,Z 55.000,A 180.000,B 0.000,C 180.000} C_DIS
LIN {X 147.911,Y 51.668,Z 55.000,A 180.000,B 0.000,C 180.000} C_DIS
LIN {X 147.846,Y 51.496,Z 55.000,A 180.000,B 0.000,C 180.000} C_DIS
LIN {X 147.299,Y 50.059,Z 55.000,A 180.000,B 0.000,C 180.000} C_DIS
LIN {X 147.227,Y 49.880,Z 55.000,A 180.000,B 0.000,C 180.000} C_DIS
LIN {X 146.645,Y 48.450,Z 55.000,A 180.000,B 0.000,C 180.000} C_DIS
LIN {X 146.595,Y 48.331,Z 55.000,A 180.000,B 0.000,C 180.000} C_DIS
LIN {X 145.947,Y 46.841,Z 55.000,A 180.000,B 0.000,C 180.000} C_DIS
LIN {X 145.880,Y 46.692,Z 55.000,A 180.000,B 0.000,C 180.000} C_DIS
LIN {X 145.203,Y 45.232,Z 55.000,A 180.000,B 0.000,C 180.000} C_DIS
LIN {X 145.164,Y 45.151,Z 55.000,A 180.000,B 0.000,C 180.000} C_DIS
LIN {X 144.449,Y 43.697,Z 55.000,A 180.000,B 0.000,C 180.000} C_DIS
LIN {X 144.413,Y 43.623,Z 55.000,A 180.000,B 0.000,C 180.000} C_DIS
LIN {X 144.320,Y 43.444,Z 55.000,A 180.000,B 0.000,C 180.000} C_DIS
LIN {X 143.668,Y 42.193,Z 55.000,A 180.000,B 0.000,C 180.000} C_DIS
LIN {X 143.574,Y 42.014,Z 55.000,A 180.000,B 0.000,C 180.000} C_DIS
LIN {X 142.785,Y 40.584,Z 55.000,A 180.000,B 0.000,C 180.000} C_DIS
LIN {X 142.683,Y 40.405,Z 55.000,A 180.000,B 0.000,C 180.000} C_DIS
LIN {X 141.947,Y 39.141,Z 55.000,A 180.000,B 0.000,C 180.000} C_DIS
LIN {X 141.849,Y 38.975,Z 55.000,A 180.000,B 0.000,C 180.000} C_DIS
LIN {X 141.768,Y 38.842,Z 55.000,A 180.000,B 0.000,C 180.000} C_DIS
LIN {X 140.971,Y 37.545,Z 55.000,A 180.000,B 0.000,C 180.000} C_DIS
LIN {X 140.874,Y 37.393,Z 55.000,A 180.000,B 0.000,C 180.000} C_DIS
LIN {X 140.047,Y 36.115,Z 55.000,A 180.000,B 0.000,C 180.000} C_DIS
LIN {X 139.980,Y 36.012,Z 55.000,A 180.000,B 0.000,C 180.000} C_DIS
LIN {X 139.928,Y 35.936,Z 55.000,A 180.000,B 0.000,C 180.000} C_DIS
LIN {X 139.076,Y 34.685,Z 55.000,A 180.000,B 0.000,C 180.000} C_DIS
LIN {X 138.953,Y 34.506,Z 55.000,A 180.000,B 0.000,C 180.000} C_DIS
LIN {X 138.014,Y 33.194,Z 55.000,A 180.000,B 0.000,C 180.000} C_DIS
LIN {X 137.927,Y 33.076,Z 55.000,A 180.000,B 0.000,C 180.000} C_DIS
LIN {X 136.941,Y 31.765,Z 55.000,A 180.000,B 0.000,C 180.000} C_DIS
LIN {X 136.848,Y 31.646,Z 55.000,A 180.000,B 0.000,C 180.000} C_DIS
LIN {X 135.861,Y 30.394,Z 55.000,A 180.000,B 0.000,C 180.000} C_DIS
LIN {X 135.714,Y 30.215,Z 55.000,A 180.000,B 0.000,C 180.000} C_DIS
LIN {X 134.796,Y 29.106,Z 55.000,A 180.000,B 0.000,C 180.000} C_DIS
LIN {X 134.677,Y 28.964,Z 55.000,A 180.000,B 0.000,C 180.000} C_DIS
LIN {X 133.590,Y 27.713,Z 55.000,A 180.000,B 0.000,C 180.000} C_DIS
LIN {X 133.544,Y 27.660,Z 55.000,A 180.000,B 0.000,C 180.000} C_DIS
LIN {X 133.430,Y 27.534,Z 55.000,A 180.000,B 0.000,C 180.000} C_DIS
LIN {X 132.453,Y 26.461,Z 55.000,A 180.000,B 0.000,C 180.000} C_DIS
LIN {X 132.293,Y 26.289,Z 55.000,A 180.000,B 0.000,C 180.000} C_DIS
LIN {X 131.220,Y 25.165,Z 55.000,A 180.000,B 0.000,C 180.000} C_DIS
LIN {X 131.090,Y 25.031,Z 55.000,A 180.000,B 0.000,C 180.000} C_DIS
LIN {X 129.969,Y 23.910,Z 55.000,A 180.000,B 0.000,C 180.000} C_DIS
LIN {X 129.835,Y 23.780,Z 55.000,A 180.000,B 0.000,C 180.000} C_DIS
LIN {X 128.711,Y 22.707,Z 55.000,A 180.000,B 0.000,C 180.000} C_DIS
LIN {X 128.539,Y 22.547,Z 55.000,A 180.000,B 0.000,C 180.000} C_DIS
LIN {X 127.466,Y 21.570,Z 55.000,A 180.000,B 0.000,C 180.000} C_DIS
LIN {X 127.340,Y 21.456,Z 55.000,A 180.000,B 0.000,C 180.000} C_DIS
LIN {X 127.287,Y 21.410,Z 55.000,A 180.000,B 0.000,C 180.000} C_DIS
LIN {X 126.036,Y 20.323,Z 55.000,A 180.000,B 0.000,C 180.000} C_DIS
LIN {X 125.894,Y 20.204,Z 55.000,A 180.000,B 0.000,C 180.000} C_DIS
LIN {X 124.785,Y 19.286,Z 55.000,A 180.000,B 0.000,C 180.000} C_DIS
LIN {X 124.606,Y 19.139,Z 55.000,A 180.000,B 0.000,C 180.000} C_DIS
LIN {X 123.354,Y 18.152,Z 55.000,A 180.000,B 0.000,C 180.000} C_DIS
LIN {X 123.235,Y 18.059,Z 55.000,A 180.000,B 0.000,C 180.000} C_DIS
LIN {X 121.924,Y 17.073,Z 55.000,A 180.000,B 0.000,C 180.000} C_DIS
LIN {X 121.806,Y 16.986,Z 55.000,A 180.000,B 0.000,C 180.000} C_DIS
LIN {X 120.494,Y 16.047,Z 55.000,A 180.000,B 0.000,C 180.000} C_DIS
LIN {X 120.315,Y 15.924,Z 55.000,A 180.000,B 0.000,C 180.000} C_DIS
LIN {X 119.064,Y 15.072,Z 55.000,A 180.000,B 0.000,C 180.000} C_DIS
LIN {X 118.988,Y 15.020,Z 55.000,A 180.000,B 0.000,C 180.000} C_DIS
LIN {X 118.885,Y 14.953,Z 55.000,A 180.000,B 0.000,C 180.000} C_DIS
LIN {X 117.607,Y 14.126,Z 55.000,A 180.000,B 0.000,C 180.000} C_DIS
LIN {X 117.455,Y 14.029,Z 55.000,A 180.000,B 0.000,C 180.000} C_DIS
LIN {X 116.158,Y 13.232,Z 55.000,A 180.000,B 0.000,C 180.000} C_DIS
LIN {X 116.025,Y 13.151,Z 55.000,A 180.000,B 0.000,C 180.000} C_DIS
LIN {X 115.859,Y 13.053,Z 55.000,A 180.000,B 0.000,C 180.000} C_DIS
LIN {X 114.595,Y 12.317,Z 55.000,A 180.000,B 0.000,C 180.000} C_DIS
LIN {X 114.416,Y 12.215,Z 55.000,A 180.000,B 0.000,C 180.000} C_DIS
LIN {X 112.986,Y 11.426,Z 55.000,A 180.000,B 0.000,C 180.000} C_DIS
LIN {X 112.807,Y 11.332,Z 55.000,A 180.000,B 0.000,C 180.000} C_DIS
LIN {X 111.556,Y 10.680,Z 55.000,A 180.000,B 0.000,C 180.000} C_DIS
LIN {X 111.377,Y 10.587,Z 55.000,A 180.000,B 0.000,C 180.000} C_DIS
LIN {X 111.303,Y 10.551,Z 55.000,A 180.000,B 0.000,C 180.000} C_DIS
LIN {X 109.849,Y 9.836,Z 55.000,A 180.000,B 0.000,C 180.000} C_DIS
LIN {X 109.768,Y 9.797,Z 55.000,A 180.000,B 0.000,C 180.000} C_DIS
LIN {X 108.308,Y 9.120,Z 55.000,A 180.000,B 0.000,C 180.000} C_DIS
LIN {X 108.159,Y 9.053,Z 55.000,A 180.000,B 0.000,C 180.000} C_DIS
LIN {X 106.669,Y 8.405,Z 55.000,A 180.000,B 0.000,C 180.000} C_DIS
LIN {X 106.550,Y 8.355,Z 55.000,A 180.000,B 0.000,C 180.000} C_DIS
LIN {X 105.120,Y 7.773,Z 55.000,A 180.000,B 0.000,C 180.000} C_DIS
LIN {X 104.941,Y 7.701,Z 55.000,A 180.000,B 0.000,C 180.000} C_DIS
LIN {X 103.504,Y 7.154,Z 55.000,A 180.000,B 0.000,C 180.000} C_DIS
LIN {X 103.332,Y 7.089,Z 55.000,A 180.000,B 0.000,C 180.000} C_DIS
LIN {X 103.153,Y 7.026,Z 55.000,A 180.000,B 0.000,C 180.000} C_DIS
LIN {X 101.723,Y 6.520,Z 55.000,A 180.000,B 0.000,C 180.000} C_DIS
LIN {X 101.545,Y 6.460,Z 55.000,A 180.000,B 0.000,C 180.000} C_DIS
LIN {X 100.114,Y 5.992,Z 55.000,A 180.000,B 0.000,C 180.000} C_DIS
LIN {X 99.936,Y 5.935,Z 55.000,A 180.000,B 0.000,C 180.000} C_DIS
LIN {X 98.505,Y 5.503,Z 55.000,A 180.000,B 0.000,C 180.000} C_DIS
LIN {X 98.327,Y 5.450,Z 55.000,A 180.000,B 0.000,C 180.000} C_DIS
LIN {X 98.148,Y 5.400,Z 55.000,A 180.000,B 0.000,C 180.000} C_DIS
LIN {X 96.718,Y 5.005,Z 55.000,A 180.000,B 0.000,C 180.000} C_DIS
LIN {X 96.539,Y 4.958,Z 55.000,A 180.000,B 0.000,C 180.000} C_DIS
LIN {X 95.109,Y 4.598,Z 55.000,A 180.000,B 0.000,C 180.000} C_DIS
LIN {X 94.930,Y 4.554,Z 55.000,A 180.000,B 0.000,C 180.000} C_DIS
LIN {X 94.751,Y 4.513,Z 55.000,A 180.000,B 0.000,C 180.000} C_DIS
LIN {X 93.321,Y 4.189,Z 55.000,A 180.000,B 0.000,C 180.000} C_DIS
LIN {X 93.142,Y 4.150,Z 55.000,A 180.000,B 0.000,C 180.000} C_DIS
LIN {X 91.533,Y 3.825,Z 55.000,A 180.000,B 0.000,C 180.000} C_DIS
LIN {X 91.355,Y 3.792,Z 55.000,A 180.000,B 0.000,C 180.000} C_DIS
LIN {X 89.925,Y 3.538,Z 55.000,A 180.000,B 0.000,C 180.000} C_DIS
LIN {X 89.746,Y 3.506,Z 55.000,A 180.000,B 0.000,C 180.000} C_DIS
LIN {X 89.567,Y 3.479,Z 55.000,A 180.000,B 0.000,C 180.000} C_DIS
LIN {X 88.137,Y 3.259,Z 55.000,A 180.000,B 0.000,C 180.000} C_DIS
LIN {X 87.958,Y 3.233,Z 55.000,A 180.000,B 0.000,C 180.000} C_DIS
LIN {X 86.349,Y 3.025,Z 55.000,A 180.000,B 0.000,C 180.000} C_DIS
LIN {X 86.170,Y 3.004,Z 55.000,A 180.000,B 0.000,C 180.000} C_DIS
LIN {X 84.561,Y 2.833,Z 55.000,A 180.000,B 0.000,C 180.000} C_DIS
LIN {X 84.383,Y 2.818,Z 55.000,A 180.000,B 0.000,C 180.000} C_DIS
LIN {X 82.952,Y 2.700,Z 55.000,A 180.000,B 0.000,C 180.000} C_DIS
LIN {X 82.774,Y 2.686,Z 55.000,A 180.000,B 0.000,C 180.000} C_DIS
LIN {X 82.761,Y 2.685,Z 55.000,A 180.000,B 0.000,C 180.000} C_DIS
LIN {X 82.595,Y 2.675,Z 55.000,A 180.000,B 0.000,C 180.000} C_DIS
LIN {X 81.165,Y 2.591,Z 55.000,A 180.000,B 0.000,C 180.000} C_DIS
LIN {X 80.986,Y 2.581,Z 55.000,A 180.000,B 0.000,C 180.000} C_DIS
LIN {X 79.377,Y 2.525,Z 55.000,A 180.000,B 0.000,C 180.000} C_DIS
LIN {X 79.198,Y 2.520,Z 55.000,A 180.000,B 0.000,C 180.000} C_DIS
LIN {X 77.589,Y 2.501,Z 55.000,A 180.000,B 0.000,C 180.000} C_DIS
LIN {X 77.411,Y 2.501,Z 55.000,A 180.000,B 0.000,C 180.000} C_DIS
LIN {X 75.802,Y 2.520,Z 55.000,A 180.000,B 0.000,C 180.000} C_DIS
LIN {X 75.623,Y 2.525,Z 55.000,A 180.000,B 0.000,C 180.000} C_DIS
LIN {X 74.014,Y 2.581,Z 55.000,A 180.000,B 0.000,C 180.000} C_DIS
LIN {X 73.835,Y 2.591,Z 55.000,A 180.000,B 0.000,C 180.000} C_DIS
LIN {X 72.405,Y 2.675,Z 55.000,A 180.000,B 0.000,C 180.000} C_DIS
LIN {X 72.239,Y 2.685,Z 55.000,A 180.000,B 0.000,C 180.000} C_DIS
LIN {X 72.226,Y 2.686,Z 55.000,A 180.000,B 0.000,C 180.000} C_DIS
LIN {X 72.048,Y 2.700,Z 55.000,A 180.000,B 0.000,C 180.000} C_DIS
LIN {X 70.617,Y 2.818,Z 55.000,A 180.000,B 0.000,C 180.000} C_DIS
LIN {X 70.439,Y 2.833,Z 55.000,A 180.000,B 0.000,C 180.000} C_DIS
LIN {X 68.830,Y 3.004,Z 55.000,A 180.000,B 0.000,C 180.000} C_DIS
LIN {X 68.651,Y 3.025,Z 55.000,A 180.000,B 0.000,C 180.000} C_DIS
LIN {X 67.042,Y 3.233,Z 55.000,A 180.000,B 0.000,C 180.000} C_DIS
LIN {X 66.863,Y 3.259,Z 55.000,A 180.000,B 0.000,C 180.000} C_DIS
LIN {X 65.433,Y 3.479,Z 55.000,A 180.000,B 0.000,C 180.000} C_DIS
LIN {X 65.254,Y 3.506,Z 55.000,A 180.000,B 0.000,C 180.000} C_DIS
LIN {X 65.075,Y 3.538,Z 55.000,A 180.000,B 0.000,C 180.000} C_DIS
LIN {X 63.645,Y 3.792,Z 55.000,A 180.000,B 0.000,C 180.000} C_DIS
LIN {X 63.467,Y 3.825,Z 55.000,A 180.000,B 0.000,C 180.000} C_DIS
LIN {X 61.858,Y 4.150,Z 55.000,A 180.000,B 0.000,C 180.000} C_DIS
LIN {X 61.679,Y 4.189,Z 55.000,A 180.000,B 0.000,C 180.000} C_DIS
LIN {X 60.249,Y 4.513,Z 55.000,A 180.000,B 0.000,C 180.000} C_DIS
LIN {X 60.070,Y 4.554,Z 55.000,A 180.000,B 0.000,C 180.000} C_DIS
LIN {X 59.891,Y 4.598,Z 55.000,A 180.000,B 0.000,C 180.000} C_DIS
LIN {X 58.461,Y 4.958,Z 55.000,A 180.000,B 0.000,C 180.000} C_DIS
LIN {X 58.282,Y 5.005,Z 55.000,A 180.000,B 0.000,C 180.000} C_DIS
LIN {X 56.852,Y 5.400,Z 55.000,A 180.000,B 0.000,C 180.000} C_DIS
LIN {X 56.673,Y 5.450,Z 55.000,A 180.000,B 0.000,C 180.000} C_DIS
LIN {X 56.495,Y 5.503,Z 55.000,A 180.000,B 0.000,C 180.000} C_DIS
LIN {X 55.064,Y 5.935,Z 55.000,A 180.000,B 0.000,C 180.000} C_DIS
LIN {X 54.886,Y 5.992,Z 55.000,A 180.000,B 0.000,C 180.000} C_DIS
LIN {X 53.455,Y 6.460,Z 55.000,A 180.000,B 0.000,C 180.000} C_DIS
LIN {X 53.277,Y 6.520,Z 55.000,A 180.000,B 0.000,C 180.000} C_DIS
LIN {X 51.847,Y 7.026,Z 55.000,A 180.000,B 0.000,C 180.000} C_DIS
LIN {X 51.668,Y 7.089,Z 55.000,A 180.000,B 0.000,C 180.000} C_DIS
LIN {X 51.496,Y 7.154,Z 55.000,A 180.000,B 0.000,C 180.000} C_DIS
LIN {X 50.059,Y 7.701,Z 55.000,A 180.000,B 0.000,C 180.000} C_DIS
LIN {X 49.880,Y 7.773,Z 55.000,A 180.000,B 0.000,C 180.000} C_DIS
LIN {X 48.450,Y 8.355,Z 55.000,A 180.000,B 0.000,C 180.000} C_DIS
LIN {X 48.331,Y 8.405,Z 55.000,A 180.000,B 0.000,C 180.000} C_DIS
LIN {X 46.841,Y 9.053,Z 55.000,A 180.000,B 0.000,C 180.000} C_DIS
LIN {X 46.692,Y 9.120,Z 55.000,A 180.000,B 0.000,C 180.000} C_DIS
LIN {X 45.232,Y 9.797,Z 55.000,A 180.000,B 0.000,C 180.000} C_DIS
LIN {X 45.151,Y 9.836,Z 55.000,A 180.000,B 0.000,C 180.000} C_DIS
LIN {X 43.697,Y 10.551,Z 55.000,A 180.000,B 0.000,C 180.000} C_DIS
LIN {X 43.623,Y 10.587,Z 55.000,A 180.000,B 0.000,C 180.000} C_DIS
LIN {X 43.444,Y 10.680,Z 55.000,A 180.000,B 0.000,C 180.000} C_DIS
LIN {X 42.193,Y 11.332,Z 55.000,A 180.000,B 0.000,C 180.000} C_DIS
LIN {X 42.014,Y 11.426,Z 55.000,A 180.000,B 0.000,C 180.000} C_DIS
LIN {X 40.584,Y 12.215,Z 55.000,A 180.000,B 0.000,C 180.000} C_DIS
LIN {X 40.405,Y 12.317,Z 55.000,A 180.000,B 0.000,C 180.000} C_DIS
LIN {X 39.141,Y 13.053,Z 55.000,A 180.000,B 0.000,C 180.000} C_DIS
LIN {X 38.975,Y 13.151,Z 55.000,A 180.000,B 0.000,C 180.000} C_DIS
LIN {X 38.842,Y 13.232,Z 55.000,A 180.000,B 0.000,C 180.000} C_DIS
LIN {X 37.545,Y 14.029,Z 55.000,A 180.000,B 0.000,C 180.000} C_DIS
LIN {X 37.393,Y 14.126,Z 55.000,A 180.000,B 0.000,C 180.000} C_DIS
LIN {X 36.115,Y 14.953,Z 55.000,A 180.000,B 0.000,C 180.000} C_DIS
LIN {X 36.012,Y 15.020,Z 55.000,A 180.000,B 0.000,C 180.000} C_DIS
LIN {X 35.936,Y 15.072,Z 55.000,A 180.000,B 0.000,C 180.000} C_DIS
LIN {X 34.685,Y 15.924,Z 55.000,A 180.000,B 0.000,C 180.000} C_DIS
LIN {X 34.506,Y 16.047,Z 55.000,A 180.000,B 0.000,C 180.000} C_DIS
LIN {X 33.194,Y 16.986,Z 55.000,A 180.000,B 0.000,C 180.000} C_DIS
LIN {X 33.076,Y 17.073,Z 55.000,A 180.000,B 0.000,C 180.000} C_DIS
LIN {X 31.765,Y 18.059,Z 55.000,A 180.000,B 0.000,C 180.000} C_DIS
LIN {X 31.646,Y 18.152,Z 55.000,A 180.000,B 0.000,C 180.000} C_DIS
LIN {X 30.394,Y 19.139,Z 55.000,A 180.000,B 0.000,C 180.000} C_DIS
LIN {X 30.215,Y 19.286,Z 55.000,A 180.000,B 0.000,C 180.000} C_DIS
LIN {X 29.106,Y 20.204,Z 55.000,A 180.000,B 0.000,C 180.000} C_DIS
LIN {X 28.964,Y 20.323,Z 55.000,A 180.000,B 0.000,C 180.000} C_DIS
LIN {X 27.713,Y 21.410,Z 55.000,A 180.000,B 0.000,C 180.000} C_DIS
LIN {X 27.660,Y 21.456,Z 55.000,A 180.000,B 0.000,C 180.000} C_DIS
LIN {X 27.534,Y 21.570,Z 55.000,A 180.000,B 0.000,C 180.000} C_DIS
LIN {X 26.461,Y 22.547,Z 55.000,A 180.000,B 0.000,C 180.000} C_DIS
LIN {X 26.289,Y 22.707,Z 55.000,A 180.000,B 0.000,C 180.000} C_DIS
LIN {X 25.165,Y 23.780,Z 55.000,A 180.000,B 0.000,C 180.000} C_DIS
LIN {X 25.031,Y 23.910,Z 55.000,A 180.000,B 0.000,C 180.000} C_DIS
LIN {X 23.910,Y 25.031,Z 55.000,A 180.000,B 0.000,C 180.000} C_DIS
LIN {X 23.780,Y 25.165,Z 55.000,A 180.000,B 0.000,C 180.000} C_DIS
LIN {X 22.707,Y 26.289,Z 55.000,A 180.000,B 0.000,C 180.000} C_DIS
LIN {X 22.547,Y 26.461,Z 55.000,A 180.000,B 0.000,C 180.000} C_DIS
LIN {X 21.570,Y 27.534,Z 55.000,A 180.000,B 0.000,C 180.000} C_DIS
LIN {X 21.456,Y 27.660,Z 55.000,A 180.000,B 0.000,C 180.000} C_DIS
LIN {X 21.410,Y 27.713,Z 55.000,A 180.000,B 0.000,C 180.000} C_DIS
LIN {X 20.323,Y 28.964,Z 55.000,A 180.000,B 0.000,C 180.000} C_DIS
LIN {X 20.204,Y 29.106,Z 55.000,A 180.000,B 0.000,C 180.000} C_DIS
LIN {X 19.286,Y 30.215,Z 55.000,A 180.000,B 0.000,C 180.000} C_DIS
LIN {X 19.139,Y 30.394,Z 55.000,A 180.000,B 0.000,C 180.000} C_DIS
LIN {X 18.152,Y 31.646,Z 55.000,A 180.000,B 0.000,C 180.000} C_DIS
LIN {X 18.059,Y 31.765,Z 55.000,A 180.000,B 0.000,C 180.000} C_DIS
LIN {X 17.073,Y 33.076,Z 55.000,A 180.000,B 0.000,C 180.000} C_DIS
LIN {X 16.986,Y 33.194,Z 55.000,A 180.000,B 0.000,C 180.000} C_DIS
LIN {X 16.047,Y 34.506,Z 55.000,A 180.000,B 0.000,C 180.000} C_DIS
LIN {X 15.924,Y 34.685,Z 55.000,A 180.000,B 0.000,C 180.000} C_DIS
LIN {X 15.072,Y 35.936,Z 55.000,A 180.000,B 0.000,C 180.000} C_DIS
LIN {X 15.020,Y 36.012,Z 55.000,A 180.000,B 0.000,C 180.000} C_DIS
LIN {X 14.953,Y 36.115,Z 55.000,A 180.000,B 0.000,C 180.000} C_DIS
LIN {X 14.126,Y 37.393,Z 55.000,A 180.000,B 0.000,C 180.000} C_DIS
LIN {X 14.029,Y 37.545,Z 55.000,A 180.000,B 0.000,C 180.000} C_DIS
LIN {X 13.232,Y 38.842,Z 55.000,A 180.000,B 0.000,C 180.000} C_DIS
LIN {X 13.151,Y 38.975,Z 55.000,A 180.000,B 0.000,C 180.000} C_DIS
LIN {X 13.053,Y 39.141,Z 55.000,A 180.000,B 0.000,C 180.000} C_DIS
LIN {X 12.317,Y 40.405,Z 55.000,A 180.000,B 0.000,C 180.000} C_DIS
LIN {X 12.215,Y 40.584,Z 55.000,A 180.000,B 0.000,C 180.000} C_DIS
LIN {X 11.426,Y 42.014,Z 55.000,A 180.000,B 0.000,C 180.000} C_DIS
LIN {X 11.332,Y 42.193,Z 55.000,A 180.000,B 0.000,C 180.000} C_DIS
LIN {X 10.680,Y 43.444,Z 55.000,A 180.000,B 0.000,C 180.000} C_DIS
LIN {X 10.587,Y 43.623,Z 55.000,A 180.000,B 0.000,C 180.000} C_DIS
LIN {X 10.551,Y 43.697,Z 55.000,A 180.000,B 0.000,C 180.000} C_DIS
LIN {X 9.836,Y 45.151,Z 55.000,A 180.000,B 0.000,C 180.000} C_DIS
LIN {X 9.797,Y 45.232,Z 55.000,A 180.000,B 0.000,C 180.000} C_DIS
LIN {X 9.120,Y 46.692,Z 55.000,A 180.000,B 0.000,C 180.000} C_DIS
LIN {X 9.053,Y 46.841,Z 55.000,A 180.000,B 0.000,C 180.000} C_DIS
LIN {X 8.405,Y 48.331,Z 55.000,A 180.000,B 0.000,C 180.000} C_DIS
LIN {X 8.355,Y 48.450,Z 55.000,A 180.000,B 0.000,C 180.000} C_DIS
LIN {X 7.773,Y 49.880,Z 55.000,A 180.000,B 0.000,C 180.000} C_DIS
LIN {X 7.701,Y 50.059,Z 55.000,A 180.000,B 0.000,C 180.000} C_DIS
LIN {X 7.154,Y 51.496,Z 55.000,A 180.000,B 0.000,C 180.000} C_DIS
LIN {X 7.089,Y 51.668,Z 55.000,A 180.000,B 0.000,C 180.000} C_DIS
LIN {X 7.026,Y 51.847,Z 55.000,A 180.000,B 0.000,C 180.000} C_DIS
LIN {X 6.520,Y 53.277,Z 55.000,A 180.000,B 0.000,C 180.000} C_DIS
LIN {X 6.460,Y 53.455,Z 55.000,A 180.000,B 0.000,C 180.000} C_DIS
LIN {X 5.992,Y 54.886,Z 55.000,A 180.000,B 0.000,C 180.000} C_DIS
LIN {X 5.935,Y 55.064,Z 55.000,A 180.000,B 0.000,C 180.000} C_DIS
LIN {X 5.503,Y 56.495,Z 55.000,A 180.000,B 0.000,C 180.000} C_DIS
LIN {X 5.450,Y 56.673,Z 55.000,A 180.000,B 0.000,C 180.000} C_DIS
LIN {X 5.400,Y 56.852,Z 55.000,A 180.000,B 0.000,C 180.000} C_DIS
LIN {X 5.005,Y 58.282,Z 55.000,A 180.000,B 0.000,C 180.000} C_DIS
LIN {X 4.958,Y 58.461,Z 55.000,A 180.000,B 0.000,C 180.000} C_DIS
LIN {X 4.598,Y 59.891,Z 55.000,A 180.000,B 0.000,C 180.000} C_DIS
LIN {X 4.554,Y 60.070,Z 55.000,A 180.000,B 0.000,C 180.000} C_DIS
LIN {X 4.513,Y 60.249,Z 55.000,A 180.000,B 0.000,C 180.000} C_DIS
LIN {X 4.189,Y 61.679,Z 55.000,A 180.000,B 0.000,C 180.000} C_DIS
LIN {X 4.150,Y 61.858,Z 55.000,A 180.000,B 0.000,C 180.000} C_DIS
LIN {X 3.825,Y 63.467,Z 55.000,A 180.000,B 0.000,C 180.000} C_DIS
LIN {X 3.792,Y 63.645,Z 55.000,A 180.000,B 0.000,C 180.000} C_DIS
LIN {X 3.538,Y 65.075,Z 55.000,A 180.000,B 0.000,C 180.000} C_DIS
LIN {X 3.506,Y 65.254,Z 55.000,A 180.000,B 0.000,C 180.000} C_DIS
LIN {X 3.479,Y 65.433,Z 55.000,A 180.000,B 0.000,C 180.000} C_DIS
LIN {X 3.259,Y 66.863,Z 55.000,A 180.000,B 0.000,C 180.000} C_DIS
LIN {X 3.233,Y 67.042,Z 55.000,A 180.000,B 0.000,C 180.000} C_DIS
LIN {X 3.025,Y 68.651,Z 55.000,A 180.000,B 0.000,C 180.000} C_DIS
LIN {X 3.004,Y 68.830,Z 55.000,A 180.000,B 0.000,C 180.000} C_DIS
LIN {X 2.833,Y 70.439,Z 55.000,A 180.000,B 0.000,C 180.000} C_DIS
LIN {X 2.818,Y 70.617,Z 55.000,A 180.000,B 0.000,C 180.000} C_DIS
LIN {X 2.700,Y 72.048,Z 55.000,A 180.000,B 0.000,C 180.000} C_DIS
LIN {X 2.686,Y 72.226,Z 55.000,A 180.000,B 0.000,C 180.000} C_DIS
LIN {X 2.685,Y 72.239,Z 55.000,A 180.000,B 0.000,C 180.000} C_DIS
LIN {X 2.675,Y 72.405,Z 55.000,A 180.000,B 0.000,C 180.000} C_DIS
LIN {X 2.591,Y 73.835,Z 55.000,A 180.000,B 0.000,C 180.000} C_DIS
LIN {X 2.581,Y 74.014,Z 55.000,A 180.000,B 0.000,C 180.000} C_DIS
LIN {X 2.525,Y 75.623,Z 55.000,A 180.000,B 0.000,C 180.000} C_DIS
LIN {X 2.520,Y 75.802,Z 55.000,A 180.000,B 0.000,C 180.000} C_DIS
LIN {X 2.506,Y 76.973,Z 55.000,A 180.000,B 0.000,C 180.000} C_DIS
LIN {X 2.501,Y 77.411,Z 55.000,A 180.000,B 0.000,C 180.000} C_DIS
LIN {X 2.501,Y 77.589,Z 55.000,A 180.000,B 0.000,C 180.000} C_DIS
LIN {X 2.520,Y 79.198,Z 55.000,A 180.000,B 0.000,C 180.000} C_DIS
LIN {X 2.525,Y 79.377,Z 55.000,A 180.000,B 0.000,C 180.000} C_DIS
LIN {X 2.581,Y 80.986,Z 55.000,A 180.000,B 0.000,C 180.000} C_DIS
LIN {X 2.591,Y 81.165,Z 55.000,A 180.000,B 0.000,C 180.000} C_DIS
LIN {X 2.675,Y 82.595,Z 55.000,A 180.000,B 0.000,C 180.000} C_DIS
LIN {X 2.685,Y 82.761,Z 55.000,A 180.000,B 0.000,C 180.000} C_DIS
LIN {X 2.686,Y 82.774,Z 55.000,A 180.000,B 0.000,C 180.000} C_DIS
LIN {X 2.700,Y 82.952,Z 55.000,A 180.000,B 0.000,C 180.000} C_DIS
LIN {X 2.818,Y 84.383,Z 55.000,A 180.000,B 0.000,C 180.000} C_DIS
LIN {X 2.833,Y 84.561,Z 55.000,A 180.000,B 0.000,C 180.000} C_DIS
LIN {X 3.004,Y 86.170,Z 55.000,A 180.000,B 0.000,C 180.000} C_DIS
LIN {X 3.025,Y 86.349,Z 55.000,A 180.000,B 0.000,C 180.000} C_DIS
LIN {X 3.233,Y 87.958,Z 55.000,A 180.000,B 0.000,C 180.000} C_DIS
LIN {X 3.259,Y 88.137,Z 55.000,A 180.000,B 0.000,C 180.000} C_DIS
LIN {X 3.479,Y 89.567,Z 55.000,A 180.000,B 0.000,C 180.000} C_DIS
LIN {X 3.506,Y 89.746,Z 55.000,A 180.000,B 0.000,C 180.000} C_DIS
LIN {X 3.538,Y 89.925,Z 55.000,A 180.000,B 0.000,C 180.000} C_DIS
LIN {X 3.792,Y 91.355,Z 55.000,A 180.000,B 0.000,C 180.000} C_DIS
LIN {X 3.825,Y 91.533,Z 55.000,A 180.000,B 0.000,C 180.000} C_DIS
LIN {X 4.150,Y 93.142,Z 55.000,A 180.000,B 0.000,C 180.000} C_DIS
LIN {X 4.189,Y 93.321,Z 55.000,A 180.000,B 0.000,C 180.000} C_DIS
LIN {X 4.513,Y 94.751,Z 55.000,A 180.000,B 0.000,C 180.000} C_DIS
LIN {X 4.554,Y 94.930,Z 55.000,A 180.000,B 0.000,C 180.000} C_DIS
LIN {X 4.598,Y 95.109,Z 55.000,A 180.000,B 0.000,C 180.000} C_DIS
LIN {X 4.958,Y 96.539,Z 55.000,A 180.000,B 0.000,C 180.000} C_DIS
LIN {X 5.005,Y 96.718,Z 55.000,A 180.000,B 0.000,C 180.000} C_DIS
LIN {X 5.400,Y 98.148,Z 55.000,A 180.000,B 0.000,C 180.000} C_DIS
LIN {X 5.450,Y 98.327,Z 55.000,A 180.000,B 0.000,C 180.000} C_DIS
LIN {X 5.503,Y 98.505,Z 55.000,A 180.000,B 0.000,C 180.000} C_DIS
LIN {X 5.935,Y 99.936,Z 55.000,A 180.000,B 0.000,C 180.000} C_DIS
LIN {X 5.992,Y 100.114,Z 55.000,A 180.000,B 0.000,C 180.000} C_DIS
LIN {X 6.460,Y 101.545,Z 55.000,A 180.000,B 0.000,C 180.000} C_DIS
LIN {X 6.520,Y 101.723,Z 55.000,A 180.000,B 0.000,C 180.000} C_DIS
LIN {X 7.026,Y 103.153,Z 55.000,A 180.000,B 0.000,C 180.000} C_DIS
LIN {X 7.089,Y 103.332,Z 55.000,A 180.000,B 0.000,C 180.000} C_DIS
LIN {X 7.154,Y 103.504,Z 55.000,A 180.000,B 0.000,C 180.000} C_DIS
LIN {X 7.701,Y 104.941,Z 55.000,A 180.000,B 0.000,C 180.000} C_DIS
LIN {X 7.773,Y 105.120,Z 55.000,A 180.000,B 0.000,C 180.000} C_DIS
LIN {X 8.355,Y 106.550,Z 55.000,A 180.000,B 0.000,C 180.000} C_DIS
LIN {X 8.405,Y 106.669,Z 55.000,A 180.000,B 0.000,C 180.000} C_DIS
LIN {X 9.053,Y 108.159,Z 55.000,A 180.000,B 0.000,C 180.000} C_DIS
LIN {X 9.120,Y 108.308,Z 55.000,A 180.000,B 0.000,C 180.000} C_DIS
LIN {X 9.797,Y 109.768,Z 55.000,A 180.000,B 0.000,C 180.000} C_DIS
LIN {X 9.836,Y 109.849,Z 55.000,A 180.000,B 0.000,C 180.000} C_DIS
LIN {X 10.551,Y 111.303,Z 55.000,A 180.000,B 0.000,C 180.000} C_DIS
LIN {X 10.587,Y 111.377,Z 55.000,A 180.000,B 0.000,C 180.000} C_DIS
LIN {X 10.680,Y 111.556,Z 55.000,A 180.000,B 0.000,C 180.000} C_DIS
LIN {X 11.332,Y 112.807,Z 55.000,A 180.000,B 0.000,C 180.000} C_DIS
LIN {X 11.426,Y 112.986,Z 55.000,A 180.000,B 0.000,C 180.000} C_DIS
LIN {X 12.215,Y 114.416,Z 55.000,A 180.000,B 0.000,C 180.000} C_DIS
LIN {X 12.317,Y 114.595,Z 55.000,A 180.000,B 0.000,C 180.000} C_DIS
LIN {X 13.053,Y 115.859,Z 55.000,A 180.000,B 0.000,C 180.000} C_DIS
LIN {X 13.151,Y 116.025,Z 55.000,A 180.000,B 0.000,C 180.000} C_DIS
LIN {X 13.232,Y 116.158,Z 55.000,A 180.000,B 0.000,C 180.000} C_DIS
LIN {X 14.029,Y 117.455,Z 55.000,A 180.000,B 0.000,C 180.000} C_DIS
LIN {X 14.126,Y 117.607,Z 55.000,A 180.000,B 0.000,C 180.000} C_DIS
LIN {X 14.953,Y 118.885,Z 55.000,A 180.000,B 0.000,C 180.000} C_DIS
LIN {X 15.020,Y 118.988,Z 55.000,A 180.000,B 0.000,C 180.000} C_DIS
LIN {X 15.072,Y 119.064,Z 55.000,A 180.000,B 0.000,C 180.000} C_DIS
LIN {X 15.924,Y 120.315,Z 55.000,A 180.000,B 0.000,C 180.000} C_DIS
LIN {X 16.047,Y 120.494,Z 55.000,A 180.000,B 0.000,C 180.000} C_DIS
LIN {X 16.986,Y 121.806,Z 55.000,A 180.000,B 0.000,C 180.000} C_DIS
LIN {X 17.073,Y 121.924,Z 55.000,A 180.000,B 0.000,C 180.000} C_DIS
LIN {X 18.059,Y 123.235,Z 55.000,A 180.000,B 0.000,C 180.000} C_DIS
LIN {X 18.152,Y 123.354,Z 55.000,A 180.000,B 0.000,C 180.000} C_DIS
LIN {X 19.139,Y 124.606,Z 55.000,A 180.000,B 0.000,C 180.000} C_DIS
LIN {X 19.286,Y 124.785,Z 55.000,A 180.000,B 0.000,C 180.000} C_DIS
LIN {X 20.204,Y 125.894,Z 55.000,A 180.000,B 0.000,C 180.000} C_DIS
LIN {X 20.323,Y 126.036,Z 55.000,A 180.000,B 0.000,C 180.000} C_DIS
LIN {X 21.410,Y 127.287,Z 55.000,A 180.000,B 0.000,C 180.000} C_DIS
LIN {X 21.456,Y 127.340,Z 55.000,A 180.000,B 0.000,C 180.000} C_DIS
LIN {X 21.570,Y 127.466,Z 55.000,A 180.000,B 0.000,C 180.000} C_DIS
LIN {X 22.547,Y 128.539,Z 55.000,A 180.000,B 0.000,C 180.000} C_DIS
LIN {X 22.707,Y 128.711,Z 55.000,A 180.000,B 0.000,C 180.000} C_DIS
LIN {X 23.780,Y 129.835,Z 55.000,A 180.000,B 0.000,C 180.000} C_DIS
LIN {X 23.910,Y 129.969,Z 55.000,A 180.000,B 0.000,C 180.000} C_DIS
LIN {X 25.031,Y 131.090,Z 55.000,A 180.000,B 0.000,C 180.000} C_DIS
LIN {X 25.165,Y 131.220,Z 55.000,A 180.000,B 0.000,C 180.000} C_DIS
LIN {X 26.289,Y 132.293,Z 55.000,A 180.000,B 0.000,C 180.000} C_DIS
LIN {X 26.461,Y 132.453,Z 55.000,A 180.000,B 0.000,C 180.000} C_DIS
LIN {X 27.534,Y 133.430,Z 55.000,A 180.000,B 0.000,C 180.000} C_DIS
LIN {X 27.660,Y 133.544,Z 55.000,A 180.000,B 0.000,C 180.000} C_DIS
LIN {X 27.713,Y 133.590,Z 55.000,A 180.000,B 0.000,C 180.000} C_DIS
LIN {X 28.964,Y 134.677,Z 55.000,A 180.000,B 0.000,C 180.000} C_DIS
LIN {X 29.106,Y 134.796,Z 55.000,A 180.000,B 0.000,C 180.000} C_DIS
LIN {X 30.215,Y 135.714,Z 55.000,A 180.000,B 0.000,C 180.000} C_DIS
LIN {X 30.394,Y 135.861,Z 55.000,A 180.000,B 0.000,C 180.000} C_DIS
LIN {X 31.646,Y 136.848,Z 55.000,A 180.000,B 0.000,C 180.000} C_DIS
LIN {X 31.765,Y 136.941,Z 55.000,A 180.000,B 0.000,C 180.000} C_DIS
LIN {X 33.076,Y 137.927,Z 55.000,A 180.000,B 0.000,C 180.000} C_DIS
LIN {X 33.194,Y 138.014,Z 55.000,A 180.000,B 0.000,C 180.000} C_DIS
LIN {X 34.506,Y 138.953,Z 55.000,A 180.000,B 0.000,C 180.000} C_DIS
LIN {X 34.685,Y 139.076,Z 55.000,A 180.000,B 0.000,C 180.000} C_DIS
LIN {X 35.936,Y 139.928,Z 55.000,A 180.000,B 0.000,C 180.000} C_DIS
LIN {X 36.012,Y 139.980,Z 55.000,A 180.000,B 0.000,C 180.000} C_DIS
LIN {X 36.115,Y 140.047,Z 55.000,A 180.000,B 0.000,C 180.000} C_DIS
LIN {X 37.393,Y 140.874,Z 55.000,A 180.000,B 0.000,C 180.000} C_DIS
LIN {X 37.545,Y 140.971,Z 55.000,A 180.000,B 0.000,C 180.000} C_DIS
LIN {X 38.842,Y 141.768,Z 55.000,A 180.000,B 0.000,C 180.000} C_DIS
LIN {X 38.975,Y 141.849,Z 55.000,A 180.000,B 0.000,C 180.000} C_DIS
LIN {X 39.141,Y 141.947,Z 55.000,A 180.000,B 0.000,C 180.000} C_DIS
LIN {X 40.405,Y 142.683,Z 55.000,A 180.000,B 0.000,C 180.000} C_DIS
LIN {X 40.584,Y 142.785,Z 55.000,A 180.000,B 0.000,C 180.000} C_DIS
LIN {X 42.014,Y 143.574,Z 55.000,A 180.000,B 0.000,C 180.000} C_DIS
LIN {X 42.193,Y 143.668,Z 55.000,A 180.000,B 0.000,C 180.000} C_DIS
LIN {X 43.444,Y 144.320,Z 55.000,A 180.000,B 0.000,C 180.000} C_DIS
LIN {X 43.623,Y 144.413,Z 55.000,A 180.000,B 0.000,C 180.000} C_DIS
LIN {X 43.697,Y 144.449,Z 55.000,A 180.000,B 0.000,C 180.000} C_DIS
LIN {X 45.151,Y 145.164,Z 55.000,A 180.000,B 0.000,C 180.000} C_DIS
LIN {X 45.232,Y 145.203,Z 55.000,A 180.000,B 0.000,C 180.000} C_DIS
LIN {X 46.692,Y 145.880,Z 55.000,A 180.000,B 0.000,C 180.000} C_DIS
LIN {X 46.841,Y 145.947,Z 55.000,A 180.000,B 0.000,C 180.000} C_DIS
LIN {X 48.331,Y 146.595,Z 55.000,A 180.000,B 0.000,C 180.000} C_DIS
LIN {X 48.450,Y 146.645,Z 55.000,A 180.000,B 0.000,C 180.000} C_DIS
LIN {X 49.880,Y 147.227,Z 55.000,A 180.000,B 0.000,C 180.000} C_DIS
LIN {X 50.059,Y 147.299,Z 55.000,A 180.000,B 0.000,C 180.000} C_DIS
LIN {X 51.496,Y 147.846,Z 55.000,A 180.000,B 0.000,C 180.000} C_DIS
LIN {X 51.668,Y 147.911,Z 55.000,A 180.000,B 0.000,C 180.000} C_DIS
LIN {X 51.847,Y 147.974,Z 55.000,A 180.000,B 0.000,C 180.000} C_DIS
LIN {X 53.277,Y 148.480,Z 55.000,A 180.000,B 0.000,C 180.000} C_DIS
LIN {X 53.455,Y 148.540,Z 55.000,A 180.000,B 0.000,C 180.000} C_DIS
LIN {X 54.290,Y 148.813,Z 55.000,A 180.000,B 0.000,C 180.000} C_DIS
LIN {X 54.886,Y 149.008,Z 55.000,A 180.000,B 0.000,C 180.000} C_DIS
LIN {X 55.064,Y 149.065,Z 55.000,A 180.000,B 0.000,C 180.000} C_DIS
LIN {X 56.495,Y 149.497,Z 55.000,A 180.000,B 0.000,C 180.000} C_DIS
LIN {X 56.673,Y 149.550,Z 55.000,A 180.000,B 0.000,C 180.000} C_DIS
LIN {X 56.852,Y 149.600,Z 55.000,A 180.000,B 0.000,C 180.000} C_DIS
LIN {X 58.282,Y 149.995,Z 55.000,A 180.000,B 0.000,C 180.000} C_DIS
LIN {X 58.461,Y 150.042,Z 55.000,A 180.000,B 0.000,C 180.000} C_DIS
LIN {X 59.891,Y 150.402,Z 55.000,A 180.000,B 0.000,C 180.000} C_DIS
LIN {X 60.070,Y 150.447,Z 55.000,A 180.000,B 0.000,C 180.000} C_DIS
LIN {X 60.249,Y 150.487,Z 55.000,A 180.000,B 0.000,C 180.000} C_DIS
LIN {X 61.679,Y 150.811,Z 55.000,A 180.000,B 0.000,C 180.000} C_DIS
LIN {X 61.858,Y 150.850,Z 55.000,A 180.000,B 0.000,C 180.000} C_DIS
LIN {X 63.467,Y 151.175,Z 55.000,A 180.000,B 0.000,C 180.000} C_DIS
LIN {X 63.645,Y 151.208,Z 55.000,A 180.000,B 0.000,C 180.000} C_DIS
LIN {X 65.075,Y 151.462,Z 55.000,A 180.000,B 0.000,C 180.000} C_DIS
LIN {X 65.254,Y 151.494,Z 55.000,A 180.000,B 0.000,C 180.000} C_DIS
LIN {X 65.433,Y 151.521,Z 55.000,A 180.000,B 0.000,C 180.000} C_DIS
LIN {X 66.863,Y 151.741,Z 55.000,A 180.000,B 0.000,C 180.000} C_DIS
LIN {X 67.042,Y 151.767,Z 55.000,A 180.000,B 0.000,C 180.000} C_DIS
LIN {X 68.651,Y 151.975,Z 55.000,A 180.000,B 0.000,C 180.000} C_DIS
LIN {X 68.830,Y 151.996,Z 55.000,A 180.000,B 0.000,C 180.000} C_DIS
LIN {X 70.439,Y 152.167,Z 55.000,A 180.000,B 0.000,C 180.000} C_DIS
LIN {X 70.617,Y 152.182,Z 55.000,A 180.000,B 0.000,C 180.000} C_DIS
LIN {X 72.048,Y 152.300,Z 55.000,A 180.000,B 0.000,C 180.000} C_DIS
LIN {X 72.226,Y 152.314,Z 55.000,A 180.000,B 0.000,C 180.000} C_DIS
LIN {X 72.239,Y 152.315,Z 55.000,A 180.000,B 0.000,C 180.000} C_DIS
LIN {X 72.405,Y 152.325,Z 55.000,A 180.000,B 0.000,C 180.000} C_DIS
LIN {X 73.835,Y 152.409,Z 55.000,A 180.000,B 0.000,C 180.000} C_DIS
LIN {X 74.014,Y 152.419,Z 55.000,A 180.000,B 0.000,C 180.000} C_DIS
LIN {X 75.623,Y 152.475,Z 55.000,A 180.000,B 0.000,C 180.000} C_DIS
LIN {X 75.802,Y 152.480,Z 55.000,A 180.000,B 0.000,C 180.000} C_DIS
LIN {X 77.411,Y 152.499,Z 55.000,A 180.000,B 0.000,C 180.000} C_DIS
LIN {X 77.589,Y 152.499,Z 55.000,A 180.000,B 0.000,C 180.000} C_DIS
LIN {X 79.198,Y 152.480,Z 55.000,A 180.000,B 0.000,C 180.000} C_DIS
LIN {X 79.377,Y 152.475,Z 55.000,A 180.000,B 0.000,C 180.000} C_DIS
LIN {X 80.986,Y 152.419,Z 55.000,A 180.000,B 0.000,C 180.000} C_DIS
LIN {X 81.165,Y 152.409,Z 55.000,A 180.000,B 0.000,C 180.000} C_DIS
LIN {X 82.595,Y 152.325,Z 55.000,A 180.000,B 0.000,C 180.000} C_DIS
LIN {X 82.761,Y 152.315,Z 55.000,A 180.000,B 0.000,C 180.000} C_DIS
LIN {X 82.774,Y 152.314,Z 55.000,A 180.000,B 0.000,C 180.000} C_DIS
LIN {X 82.952,Y 152.300,Z 55.000,A 180.000,B 0.000,C 180.000} C_DIS
LIN {X 84.383,Y 152.182,Z 55.000,A 180.000,B 0.000,C 180.000} C_DIS
LIN {X 84.561,Y 152.167,Z 55.000,A 180.000,B 0.000,C 180.000} C_DIS
LIN {X 86.170,Y 151.996,Z 55.000,A 180.000,B 0.000,C 180.000} C_DIS
LIN {X 86.349,Y 151.975,Z 55.000,A 180.000,B 0.000,C 180.000} C_DIS
LIN {X 87.958,Y 151.767,Z 55.000,A 180.000,B 0.000,C 180.000} C_DIS
LIN {X 88.137,Y 151.741,Z 55.000,A 180.000,B 0.000,C 180.000} C_DIS
LIN {X 88.812,Y 151.637,Z 55.000,A 180.000,B 0.000,C 180.000} C_DIS
; Link Move Starts
LIN {X 89.123,Y 151.589,Z 55.000,A 180.000,B 0.000,C 180.000} C_DIS
LIN {X 89.434,Y 151.541,Z 54.999,A 180.000,B 0.000,C 180.000} C_DIS
LIN {X 89.746,Y 151.493,Z 54.998,A 180.000,B 0.000,C 180.000} C_DIS
LIN {X 90.056,Y 151.439,Z 54.996,A 180.000,B 0.000,C 180.000} C_DIS
LIN {X 90.366,Y 151.384,Z 54.994,A 180.000,B 0.000,C 180.000} C_DIS
LIN {X 90.676,Y 151.328,Z 54.991,A 180.000,B 0.000,C 180.000} C_DIS
LIN {X 90.986,Y 151.273,Z 54.988,A 180.000,B 0.000,C 180.000} C_DIS
LIN {X 91.297,Y 151.218,Z 54.985,A 180.000,B 0.000,C 180.000} C_DIS
LIN {X 91.606,Y 151.160,Z 54.981,A 180.000,B 0.000,C 180.000} C_DIS
LIN {X 91.915,Y 151.098,Z 54.977,A 180.000,B 0.000,C 180.000} C_DIS
LIN {X 92.224,Y 151.036,Z 54.972,A 180.000,B 0.000,C 180.000} C_DIS
LIN {X 92.378,Y 151.004,Z 54.969,A 180.000,B 0.000,C 180.000} C_DIS
LIN {X 92.532,Y 150.973,Z 54.967,A 180.000,B 0.000,C 180.000} C_DIS
LIN {X 92.687,Y 150.942,Z 54.964,A 180.000,B 0.000,C 180.000} C_DIS
LIN {X 92.841,Y 150.911,Z 54.961,A 180.000,B 0.000,C 180.000} C_DIS
LIN {X 92.996,Y 150.880,Z 54.959,A 180.000,B 0.000,C 180.000} C_DIS
LIN {X 93.150,Y 150.849,Z 54.956,A 180.000,B 0.000,C 180.000} C_DIS
LIN {X 93.304,Y 150.815,Z 54.952,A 180.000,B 0.000,C 180.000} C_DIS
LIN {X 93.457,Y 150.780,Z 54.949,A 180.000,B 0.000,C 180.000} C_DIS
LIN {X 93.611,Y 150.745,Z 54.946,A 180.000,B 0.000,C 180.000} C_DIS
LIN {X 93.765,Y 150.711,Z 54.943,A 180.000,B 0.000,C 180.000} C_DIS
LIN {X 93.918,Y 150.676,Z 54.939,A 180.000,B 0.000,C 180.000} C_DIS
LIN {X 94.072,Y 150.641,Z 54.936,A 180.000,B 0.000,C 180.000} C_DIS
LIN {X 94.226,Y 150.606,Z 54.932,A 180.000,B 0.000,C 180.000} C_DIS
LIN {X 94.379,Y 150.572,Z 54.928,A 180.000,B 0.000,C 180.000} C_DIS
LIN {X 94.533,Y 150.537,Z 54.925,A 180.000,B 0.000,C 180.000} C_DIS
LIN {X 94.686,Y 150.502,Z 54.921,A 180.000,B 0.000,C 180.000} C_DIS
LIN {X 94.840,Y 150.467,Z 54.917,A 180.000,B 0.000,C 180.000} C_DIS
LIN {X 94.993,Y 150.431,Z 54.913,A 180.000,B 0.000,C 180.000} C_DIS
LIN {X 95.146,Y 150.392,Z 54.909,A 180.000,B 0.000,C 180.000} C_DIS
LIN {X 95.299,Y 150.354,Z 54.905,A 180.000,B 0.000,C 180.000} C_DIS
LIN {X 95.451,Y 150.316,Z 54.900,A 180.000,B 0.000,C 180.000} C_DIS
LIN {X 95.604,Y 150.277,Z 54.896,A 180.000,B 0.000,C 180.000} C_DIS
LIN {X 95.757,Y 150.239,Z 54.892,A 180.000,B 0.000,C 180.000} C_DIS
LIN {X 95.910,Y 150.200,Z 54.887,A 180.000,B 0.000,C 180.000} C_DIS
LIN {X 96.062,Y 150.162,Z 54.883,A 180.000,B 0.000,C 180.000} C_DIS
LIN {X 96.215,Y 150.124,Z 54.878,A 180.000,B 0.000,C 180.000} C_DIS
LIN {X 96.368,Y 150.085,Z 54.873,A 180.000,B 0.000,C 180.000} C_DIS
LIN {X 96.521,Y 150.047,Z 54.869,A 180.000,B 0.000,C 180.000} C_DIS
LIN {X 96.673,Y 150.007,Z 54.864,A 180.000,B 0.000,C 180.000} C_DIS
LIN {X 96.825,Y 149.966,Z 54.859,A 180.000,B 0.000,C 180.000} C_DIS
LIN {X 96.977,Y 149.924,Z 54.854,A 180.000,B 0.000,C 180.000} C_DIS
LIN {X 97.053,Y 149.903,Z 54.851,A 180.000,B 0.000,C 180.000} C_DIS
LIN {X 97.129,Y 149.882,Z 54.849,A 180.000,B 0.000,C 180.000} C_DIS
LIN {X 97.205,Y 149.861,Z 54.846,A 180.000,B 0.000,C 180.000} C_DIS
LIN {X 97.280,Y 149.840,Z 54.844,A 180.000,B 0.000,C 180.000} C_DIS
LIN {X 97.356,Y 149.819,Z 54.841,A 180.000,B 0.000,C 180.000} C_DIS
LIN {X 97.432,Y 149.798,Z 54.839,A 180.000,B 0.000,C 180.000} C_DIS
LIN {X 97.508,Y 149.777,Z 54.836,A 180.000,B 0.000,C 180.000} C_DIS
LIN {X 97.660,Y 149.735,Z 54.831,A 180.000,B 0.000,C 180.000} C_DIS
LIN {X 97.812,Y 149.693,Z 54.825,A 180.000,B 0.000,C 180.000} C_DIS
LIN {X 97.964,Y 149.651,Z 54.820,A 180.000,B 0.000,C 180.000} C_DIS
LIN {X 98.115,Y 149.609,Z 54.815,A 180.000,B 0.000,C 180.000} C_DIS
LIN {X 98.267,Y 149.567,Z 54.809,A 180.000,B 0.000,C 180.000} C_DIS
LIN {X 98.343,Y 149.546,Z 54.806,A 180.000,B 0.000,C 180.000} C_DIS
LIN {X 98.418,Y 149.523,Z 54.804,A 180.000,B 0.000,C 180.000} C_DIS
LIN {X 98.569,Y 149.477,Z 54.798,A 180.000,B 0.000,C 180.000} C_DIS
LIN {X 98.645,Y 149.455,Z 54.796,A 180.000,B 0.000,C 180.000} C_DIS
LIN {X 98.795,Y 149.409,Z 54.790,A 180.000,B 0.000,C 180.000} C_DIS
LIN {X 99.021,Y 149.341,Z 54.782,A 180.000,B 0.000,C 180.000} C_DIS
LIN {X 99.172,Y 149.295,Z 54.776,A 180.000,B 0.000,C 180.000} C_DIS
LIN {X 99.248,Y 149.273,Z 54.774,A 180.000,B 0.000,C 180.000} C_DIS
LIN {X 99.398,Y 149.227,Z 54.768,A 180.000,B 0.000,C 180.000} C_DIS
LIN {X 99.625,Y 149.159,Z 54.760,A 180.000,B 0.000,C 180.000} C_DIS
LIN {X 99.775,Y 149.113,Z 54.754,A 180.000,B 0.000,C 180.000} C_DIS
LIN {X 99.851,Y 149.091,Z 54.752,A 180.000,B 0.000,C 180.000} C_DIS
LIN {X 99.926,Y 149.068,Z 54.749,A 180.000,B 0.000,C 180.000} C_DIS
LIN {X 100.002,Y 149.045,Z 54.746,A 180.000,B 0.000,C 180.000} C_DIS
LIN {X 100.076,Y 149.021,Z 54.743,A 180.000,B 0.000,C 180.000} C_DIS
LIN {X 100.151,Y 148.996,Z 54.741,A 180.000,B 0.000,C 180.000} C_DIS
LIN {X 100.301,Y 148.947,Z 54.735,A 180.000,B 0.000,C 180.000} C_DIS
LIN {X 100.525,Y 148.874,Z 54.727,A 180.000,B 0.000,C 180.000} C_DIS
LIN {X 100.675,Y 148.825,Z 54.721,A 180.000,B 0.000,C 180.000} C_DIS
LIN {X 100.750,Y 148.800,Z 54.719,A 180.000,B 0.000,C 180.000} C_DIS
LIN {X 100.900,Y 148.751,Z 54.713,A 180.000,B 0.000,C 180.000} C_DIS
LIN {X 101.349,Y 148.604,Z 54.697,A 180.000,B 0.000,C 180.000} C_DIS
LIN {X 101.498,Y 148.555,Z 54.691,A 180.000,B 0.000,C 180.000} C_DIS
LIN {X 101.648,Y 148.506,Z 54.686,A 180.000,B 0.000,C 180.000} C_DIS
LIN {X 101.723,Y 148.480,Z 54.683,A 180.000,B 0.000,C 180.000} C_DIS
LIN {X 101.871,Y 148.428,Z 54.677,A 180.000,B 0.000,C 180.000} C_DIS
LIN {X 101.945,Y 148.402,Z 54.675,A 180.000,B 0.000,C 180.000} C_DIS
LIN {X 102.094,Y 148.349,Z 54.669,A 180.000,B 0.000,C 180.000} C_DIS
LIN {X 102.613,Y 148.165,Z 54.650,A 180.000,B 0.000,C 180.000} C_DIS
LIN {X 103.059,Y 148.008,Z 54.633,A 180.000,B 0.000,C 180.000} C_DIS
LIN {X 103.207,Y 147.955,Z 54.628,A 180.000,B 0.000,C 180.000} C_DIS
LIN {X 103.282,Y 147.929,Z 54.625,A 180.000,B 0.000,C 180.000} C_DIS
LIN {X 103.356,Y 147.902,Z 54.622,A 180.000,B 0.000,C 180.000} C_DIS
LIN {X 103.503,Y 147.846,Z 54.617,A 180.000,B 0.000,C 180.000} C_DIS
LIN {X 103.945,Y 147.678,Z 54.600,A 180.000,B 0.000,C 180.000} C_DIS
LIN {X 104.165,Y 147.594,Z 54.592,A 180.000,B 0.000,C 180.000} C_DIS
LIN {X 104.901,Y 147.314,Z 54.565,A 180.000,B 0.000,C 180.000} C_DIS
LIN {X 104.975,Y 147.286,Z 54.562,A 180.000,B 0.000,C 180.000} C_DIS
LIN {X 105.048,Y 147.257,Z 54.559,A 180.000,B 0.000,C 180.000} C_DIS
LIN {X 106.507,Y 146.663,Z 54.504,A 180.000,B 0.000,C 180.000} C_DIS
LIN {X 106.580,Y 146.633,Z 54.501,A 180.000,B 0.000,C 180.000} C_DIS
LIN {X 106.652,Y 146.602,Z 54.499,A 180.000,B 0.000,C 180.000} C_DIS
LIN {X 108.169,Y 145.942,Z 54.441,A 180.000,B 0.000,C 180.000} C_DIS
LIN {X 108.241,Y 145.911,Z 54.438,A 180.000,B 0.000,C 180.000} C_DIS
LIN {X 108.455,Y 145.811,Z 54.430,A 180.000,B 0.000,C 180.000} C_DIS
LIN {X 109.455,Y 145.348,Z 54.391,A 180.000,B 0.000,C 180.000} C_DIS
LIN {X 109.598,Y 145.282,Z 54.386,A 180.000,B 0.000,C 180.000} C_DIS
LIN {X 109.741,Y 145.216,Z 54.380,A 180.000,B 0.000,C 180.000} C_DIS
LIN {X 109.813,Y 145.182,Z 54.378,A 180.000,B 0.000,C 180.000} C_DIS
LIN {X 109.883,Y 145.148,Z 54.375,A 180.000,B 0.000,C 180.000} C_DIS
LIN {X 110.307,Y 144.939,Z 54.358,A 180.000,B 0.000,C 180.000} C_DIS
LIN {X 110.449,Y 144.870,Z 54.353,A 180.000,B 0.000,C 180.000} C_DIS
LIN {X 110.873,Y 144.661,Z 54.336,A 180.000,B 0.000,C 180.000} C_DIS
LIN {X 110.943,Y 144.626,Z 54.334,A 180.000,B 0.000,C 180.000} C_DIS
LIN {X 111.085,Y 144.557,Z 54.328,A 180.000,B 0.000,C 180.000} C_DIS
LIN {X 111.367,Y 144.418,Z 54.317,A 180.000,B 0.000,C 180.000} C_DIS
LIN {X 111.437,Y 144.382,Z 54.314,A 180.000,B 0.000,C 180.000} C_DIS
LIN {X 111.507,Y 144.346,Z 54.312,A 180.000,B 0.000,C 180.000} C_DIS
LIN {X 111.647,Y 144.273,Z 54.306,A 180.000,B 0.000,C 180.000} C_DIS
LIN {X 112.066,Y 144.054,Z 54.290,A 180.000,B 0.000,C 180.000} C_DIS
LIN {X 112.206,Y 143.981,Z 54.284,A 180.000,B 0.000,C 180.000} C_DIS
LIN {X 112.415,Y 143.872,Z 54.276,A 180.000,B 0.000,C 180.000} C_DIS
LIN {X 112.555,Y 143.799,Z 54.270,A 180.000,B 0.000,C 180.000} C_DIS
LIN {X 112.624,Y 143.763,Z 54.268,A 180.000,B 0.000,C 180.000} C_DIS
LIN {X 112.764,Y 143.690,Z 54.262,A 180.000,B 0.000,C 180.000} C_DIS
LIN {X 112.904,Y 143.617,Z 54.257,A 180.000,B 0.000,C 180.000} C_DIS
LIN {X 112.973,Y 143.580,Z 54.254,A 180.000,B 0.000,C 180.000} C_DIS
LIN {X 113.111,Y 143.504,Z 54.248,A 180.000,B 0.000,C 180.000} C_DIS
LIN {X 113.180,Y 143.466,Z 54.246,A 180.000,B 0.000,C 180.000} C_DIS
LIN {X 113.318,Y 143.390,Z 54.240,A 180.000,B 0.000,C 180.000} C_DIS
LIN {X 113.525,Y 143.276,Z 54.232,A 180.000,B 0.000,C 180.000} C_DIS
LIN {X 113.663,Y 143.200,Z 54.226,A 180.000,B 0.000,C 180.000} C_DIS
LIN {X 113.732,Y 143.162,Z 54.224,A 180.000,B 0.000,C 180.000} C_DIS
LIN {X 113.870,Y 143.086,Z 54.218,A 180.000,B 0.000,C 180.000} C_DIS
LIN {X 114.077,Y 142.972,Z 54.210,A 180.000,B 0.000,C 180.000} C_DIS
LIN {X 114.215,Y 142.896,Z 54.204,A 180.000,B 0.000,C 180.000} C_DIS
LIN {X 114.284,Y 142.858,Z 54.202,A 180.000,B 0.000,C 180.000} C_DIS
LIN {X 114.421,Y 142.782,Z 54.196,A 180.000,B 0.000,C 180.000} C_DIS
LIN {X 114.490,Y 142.744,Z 54.193,A 180.000,B 0.000,C 180.000} C_DIS
LIN {X 114.558,Y 142.704,Z 54.191,A 180.000,B 0.000,C 180.000} C_DIS
LIN {X 114.695,Y 142.625,Z 54.185,A 180.000,B 0.000,C 180.000} C_DIS
LIN {X 114.831,Y 142.545,Z 54.180,A 180.000,B 0.000,C 180.000} C_DIS
LIN {X 114.967,Y 142.466,Z 54.174,A 180.000,B 0.000,C 180.000} C_DIS
LIN {X 115.103,Y 142.387,Z 54.169,A 180.000,B 0.000,C 180.000} C_DIS
LIN {X 115.239,Y 142.308,Z 54.164,A 180.000,B 0.000,C 180.000} C_DIS
LIN {X 115.307,Y 142.268,Z 54.161,A 180.000,B 0.000,C 180.000} C_DIS
LIN {X 115.375,Y 142.228,Z 54.159,A 180.000,B 0.000,C 180.000} C_DIS
LIN {X 115.443,Y 142.189,Z 54.156,A 180.000,B 0.000,C 180.000} C_DIS
LIN {X 115.511,Y 142.149,Z 54.154,A 180.000,B 0.000,C 180.000} C_DIS
LIN {X 115.579,Y 142.109,Z 54.151,A 180.000,B 0.000,C 180.000} C_DIS
LIN {X 115.647,Y 142.070,Z 54.148,A 180.000,B 0.000,C 180.000} C_DIS
LIN {X 115.783,Y 141.991,Z 54.143,A 180.000,B 0.000,C 180.000} C_DIS
LIN {X 115.919,Y 141.911,Z 54.139,A 180.000,B 0.000,C 180.000} C_DIS
LIN {X 116.055,Y 141.831,Z 54.134,A 180.000,B 0.000,C 180.000} C_DIS
LIN {X 116.189,Y 141.748,Z 54.129,A 180.000,B 0.000,C 180.000} C_DIS
LIN {X 116.323,Y 141.666,Z 54.124,A 180.000,B 0.000,C 180.000} C_DIS
LIN {X 116.457,Y 141.584,Z 54.120,A 180.000,B 0.000,C 180.000} C_DIS
LIN {X 116.592,Y 141.501,Z 54.115,A 180.000,B 0.000,C 180.000} C_DIS
LIN {X 116.726,Y 141.419,Z 54.110,A 180.000,B 0.000,C 180.000} C_DIS
LIN {X 116.860,Y 141.336,Z 54.106,A 180.000,B 0.000,C 180.000} C_DIS
LIN {X 116.994,Y 141.254,Z 54.102,A 180.000,B 0.000,C 180.000} C_DIS
LIN {X 117.128,Y 141.171,Z 54.097,A 180.000,B 0.000,C 180.000} C_DIS
LIN {X 117.263,Y 141.089,Z 54.093,A 180.000,B 0.000,C 180.000} C_DIS
LIN {X 117.397,Y 141.006,Z 54.089,A 180.000,B 0.000,C 180.000} C_DIS
LIN {X 117.531,Y 140.923,Z 54.085,A 180.000,B 0.000,C 180.000} C_DIS
LIN {X 117.663,Y 140.838,Z 54.081,A 180.000,B 0.000,C 180.000} C_DIS
LIN {X 117.795,Y 140.752,Z 54.077,A 180.000,B 0.000,C 180.000} C_DIS
LIN {X 117.927,Y 140.667,Z 54.073,A 180.000,B 0.000,C 180.000} C_DIS
LIN {X 118.060,Y 140.581,Z 54.070,A 180.000,B 0.000,C 180.000} C_DIS
LIN {X 118.192,Y 140.496,Z 54.066,A 180.000,B 0.000,C 180.000} C_DIS
LIN {X 118.324,Y 140.410,Z 54.062,A 180.000,B 0.000,C 180.000} C_DIS
LIN {X 118.456,Y 140.324,Z 54.059,A 180.000,B 0.000,C 180.000} C_DIS
LIN {X 118.588,Y 140.239,Z 54.056,A 180.000,B 0.000,C 180.000} C_DIS
LIN {X 118.721,Y 140.153,Z 54.052,A 180.000,B 0.000,C 180.000} C_DIS
LIN {X 118.853,Y 140.068,Z 54.049,A 180.000,B 0.000,C 180.000} C_DIS
LIN {X 118.985,Y 139.982,Z 54.046,A 180.000,B 0.000,C 180.000} C_DIS
LIN {X 119.115,Y 139.893,Z 54.043,A 180.000,B 0.000,C 180.000} C_DIS
LIN {X 119.245,Y 139.805,Z 54.040,A 180.000,B 0.000,C 180.000} C_DIS
LIN {X 119.376,Y 139.716,Z 54.037,A 180.000,B 0.000,C 180.000} C_DIS
LIN {X 119.506,Y 139.628,Z 54.034,A 180.000,B 0.000,C 180.000} C_DIS
LIN {X 119.636,Y 139.539,Z 54.032,A 180.000,B 0.000,C 180.000} C_DIS
LIN {X 119.766,Y 139.450,Z 54.029,A 180.000,B 0.000,C 180.000} C_DIS
LIN {X 119.896,Y 139.362,Z 54.027,A 180.000,B 0.000,C 180.000} C_DIS
LIN {X 120.157,Y 139.184,Z 54.022,A 180.000,B 0.000,C 180.000} C_DIS
LIN {X 120.417,Y 139.007,Z 54.018,A 180.000,B 0.000,C 180.000} C_DIS
LIN {X 120.674,Y 138.824,Z 54.014,A 180.000,B 0.000,C 180.000} C_DIS
LIN {X 120.930,Y 138.641,Z 54.011,A 180.000,B 0.000,C 180.000} C_DIS
LIN {X 121.186,Y 138.457,Z 54.008,A 180.000,B 0.000,C 180.000} C_DIS
LIN {X 121.442,Y 138.274,Z 54.005,A 180.000,B 0.000,C 180.000} C_DIS
LIN {X 121.698,Y 138.091,Z 54.003,A 180.000,B 0.000,C 180.000} C_DIS
LIN {X 121.953,Y 137.905,Z 54.002,A 180.000,B 0.000,C 180.000} C_DIS
LIN {X 122.205,Y 137.716,Z 54.001,A 180.000,B 0.000,C 180.000} C_DIS
LIN {X 122.456,Y 137.527,Z 54.000,A 180.000,B 0.000,C 180.000} C_DIS
LIN {X 122.641,Y 137.388,Z 54.000,A 180.000,B 0.000,C 180.000} C_DIS
; Cutting Move Starts
LIN {X 123.235,Y 136.941,Z 54.000,A 180.000,B 0.000,C 180.000} C_DIS
LIN {X 123.354,Y 136.848,Z 54.000,A 180.000,B 0.000,C 180.000} C_DIS
LIN {X 124.606,Y 135.861,Z 54.000,A 180.000,B 0.000,C 180.000} C_DIS
LIN {X 124.785,Y 135.714,Z 54.000,A 180.000,B 0.000,C 180.000} C_DIS
LIN {X 125.894,Y 134.796,Z 54.000,A 180.000,B 0.000,C 180.000} C_DIS
LIN {X 126.036,Y 134.677,Z 54.000,A 180.000,B 0.000,C 180.000} C_DIS
LIN {X 127.287,Y 133.590,Z 54.000,A 180.000,B 0.000,C 180.000} C_DIS
LIN {X 127.340,Y 133.544,Z 54.000,A 180.000,B 0.000,C 180.000} C_DIS
LIN {X 127.466,Y 133.430,Z 54.000,A 180.000,B 0.000,C 180.000} C_DIS
LIN {X 128.539,Y 132.453,Z 54.000,A 180.000,B 0.000,C 180.000} C_DIS
LIN {X 128.711,Y 132.293,Z 54.000,A 180.000,B 0.000,C 180.000} C_DIS
LIN {X 129.835,Y 131.220,Z 54.000,A 180.000,B 0.000,C 180.000} C_DIS
LIN {X 129.969,Y 131.090,Z 54.000,A 180.000,B 0.000,C 180.000} C_DIS
LIN {X 131.090,Y 129.969,Z 54.000,A 180.000,B 0.000,C 180.000} C_DIS
LIN {X 131.220,Y 129.835,Z 54.000,A 180.000,B 0.000,C 180.000} C_DIS
LIN {X 132.293,Y 128.711,Z 54.000,A 180.000,B 0.000,C 180.000} C_DIS
LIN {X 132.453,Y 128.539,Z 54.000,A 180.000,B 0.000,C 180.000} C_DIS
LIN {X 133.430,Y 127.466,Z 54.000,A 180.000,B 0.000,C 180.000} C_DIS
LIN {X 133.544,Y 127.340,Z 54.000,A 180.000,B 0.000,C 180.000} C_DIS
LIN {X 133.590,Y 127.287,Z 54.000,A 180.000,B 0.000,C 180.000} C_DIS
LIN {X 134.677,Y 126.036,Z 54.000,A 180.000,B 0.000,C 180.000} C_DIS
LIN {X 134.796,Y 125.894,Z 54.000,A 180.000,B 0.000,C 180.000} C_DIS
LIN {X 135.714,Y 124.785,Z 54.000,A 180.000,B 0.000,C 180.000} C_DIS
LIN {X 135.861,Y 124.606,Z 54.000,A 180.000,B 0.000,C 180.000} C_DIS
LIN {X 136.848,Y 123.354,Z 54.000,A 180.000,B 0.000,C 180.000} C_DIS
LIN {X 136.941,Y 123.235,Z 54.000,A 180.000,B 0.000,C 180.000} C_DIS
LIN {X 137.927,Y 121.924,Z 54.000,A 180.000,B 0.000,C 180.000} C_DIS
LIN {X 138.014,Y 121.806,Z 54.000,A 180.000,B 0.000,C 180.000} C_DIS
LIN {X 138.953,Y 120.494,Z 54.000,A 180.000,B 0.000,C 180.000} C_DIS
LIN {X 139.076,Y 120.315,Z 54.000,A 180.000,B 0.000,C 180.000} C_DIS
LIN {X 139.928,Y 119.064,Z 54.000,A 180.000,B 0.000,C 180.000} C_DIS
LIN {X 139.980,Y 118.988,Z 54.000,A 180.000,B 0.000,C 180.000} C_DIS
LIN {X 140.047,Y 118.885,Z 54.000,A 180.000,B 0.000,C 180.000} C_DIS
LIN {X 140.874,Y 117.607,Z 54.000,A 180.000,B 0.000,C 180.000} C_DIS
LIN {X 140.971,Y 117.455,Z 54.000,A 180.000,B 0.000,C 180.000} C_DIS
LIN {X 141.768,Y 116.158,Z 54.000,A 180.000,B 0.000,C 180.000} C_DIS
LIN {X 141.849,Y 116.025,Z 54.000,A 180.000,B 0.000,C 180.000} C_DIS
LIN {X 141.947,Y 115.859,Z 54.000,A 180.000,B 0.000,C 180.000} C_DIS
LIN {X 142.683,Y 114.595,Z 54.000,A 180.000,B 0.000,C 180.000} C_DIS
LIN {X 142.785,Y 114.416,Z 54.000,A 180.000,B 0.000,C 180.000} C_DIS
LIN {X 143.574,Y 112.986,Z 54.000,A 180.000,B 0.000,C 180.000} C_DIS
LIN {X 143.668,Y 112.807,Z 54.000,A 180.000,B 0.000,C 180.000} C_DIS
LIN {X 144.320,Y 111.556,Z 54.000,A 180.000,B 0.000,C 180.000} C_DIS
LIN {X 144.413,Y 111.377,Z 54.000,A 180.000,B 0.000,C 180.000} C_DIS
LIN {X 144.449,Y 111.303,Z 54.000,A 180.000,B 0.000,C 180.000} C_DIS
LIN {X 145.164,Y 109.849,Z 54.000,A 180.000,B 0.000,C 180.000} C_DIS
LIN {X 145.203,Y 109.768,Z 54.000,A 180.000,B 0.000,C 180.000} C_DIS
LIN {X 145.880,Y 108.308,Z 54.000,A 180.000,B 0.000,C 180.000} C_DIS
LIN {X 145.947,Y 108.159,Z 54.000,A 180.000,B 0.000,C 180.000} C_DIS
LIN {X 146.595,Y 106.669,Z 54.000,A 180.000,B 0.000,C 180.000} C_DIS
LIN {X 146.645,Y 106.550,Z 54.000,A 180.000,B 0.000,C 180.000} C_DIS
LIN {X 147.227,Y 105.120,Z 54.000,A 180.000,B 0.000,C 180.000} C_DIS
LIN {X 147.299,Y 104.941,Z 54.000,A 180.000,B 0.000,C 180.000} C_DIS
LIN {X 147.846,Y 103.504,Z 54.000,A 180.000,B 0.000,C 180.000} C_DIS
LIN {X 147.911,Y 103.332,Z 54.000,A 180.000,B 0.000,C 180.000} C_DIS
LIN {X 147.974,Y 103.153,Z 54.000,A 180.000,B 0.000,C 180.000} C_DIS
LIN {X 148.480,Y 101.723,Z 54.000,A 180.000,B 0.000,C 180.000} C_DIS
LIN {X 148.540,Y 101.545,Z 54.000,A 180.000,B 0.000,C 180.000} C_DIS
LIN {X 149.008,Y 100.114,Z 54.000,A 180.000,B 0.000,C 180.000} C_DIS
LIN {X 149.065,Y 99.936,Z 54.000,A 180.000,B 0.000,C 180.000} C_DIS
LIN {X 149.497,Y 98.505,Z 54.000,A 180.000,B 0.000,C 180.000} C_DIS
LIN {X 149.550,Y 98.327,Z 54.000,A 180.000,B 0.000,C 180.000} C_DIS
LIN {X 149.600,Y 98.148,Z 54.000,A 180.000,B 0.000,C 180.000} C_DIS
LIN {X 149.995,Y 96.718,Z 54.000,A 180.000,B 0.000,C 180.000} C_DIS
LIN {X 150.042,Y 96.539,Z 54.000,A 180.000,B 0.000,C 180.000} C_DIS
LIN {X 150.402,Y 95.109,Z 54.000,A 180.000,B 0.000,C 180.000} C_DIS
LIN {X 150.447,Y 94.930,Z 54.000,A 180.000,B 0.000,C 180.000} C_DIS
LIN {X 150.487,Y 94.751,Z 54.000,A 180.000,B 0.000,C 180.000} C_DIS
LIN {X 150.811,Y 93.321,Z 54.000,A 180.000,B 0.000,C 180.000} C_DIS
LIN {X 150.850,Y 93.142,Z 54.000,A 180.000,B 0.000,C 180.000} C_DIS
LIN {X 151.175,Y 91.533,Z 54.000,A 180.000,B 0.000,C 180.000} C_DIS
LIN {X 151.208,Y 91.355,Z 54.000,A 180.000,B 0.000,C 180.000} C_DIS
LIN {X 151.462,Y 89.925,Z 54.000,A 180.000,B 0.000,C 180.000} C_DIS
LIN {X 151.494,Y 89.746,Z 54.000,A 180.000,B 0.000,C 180.000} C_DIS
LIN {X 151.521,Y 89.567,Z 54.000,A 180.000,B 0.000,C 180.000} C_DIS
LIN {X 151.741,Y 88.137,Z 54.000,A 180.000,B 0.000,C 180.000} C_DIS
LIN {X 151.767,Y 87.958,Z 54.000,A 180.000,B 0.000,C 180.000} C_DIS
LIN {X 151.975,Y 86.349,Z 54.000,A 180.000,B 0.000,C 180.000} C_DIS
LIN {X 151.996,Y 86.170,Z 54.000,A 180.000,B 0.000,C 180.000} C_DIS
LIN {X 152.167,Y 84.561,Z 54.000,A 180.000,B 0.000,C 180.000} C_DIS
LIN {X 152.182,Y 84.383,Z 54.000,A 180.000,B 0.000,C 180.000} C_DIS
LIN {X 152.300,Y 82.952,Z 54.000,A 180.000,B 0.000,C 180.000} C_DIS
LIN {X 152.314,Y 82.774,Z 54.000,A 180.000,B 0.000,C 180.000} C_DIS
LIN {X 152.315,Y 82.761,Z 54.000,A 180.000,B 0.000,C 180.000} C_DIS
LIN {X 152.325,Y 82.595,Z 54.000,A 180.000,B 0.000,C 180.000} C_DIS
LIN {X 152.409,Y 81.165,Z 54.000,A 180.000,B 0.000,C 180.000} C_DIS
LIN {X 152.419,Y 80.986,Z 54.000,A 180.000,B 0.000,C 180.000} C_DIS
LIN {X 152.475,Y 79.377,Z 54.000,A 180.000,B 0.000,C 180.000} C_DIS
LIN {X 152.480,Y 79.198,Z 54.000,A 180.000,B 0.000,C 180.000} C_DIS
LIN {X 152.499,Y 77.589,Z 54.000,A 180.000,B 0.000,C 180.000} C_DIS
LIN {X 152.499,Y 77.411,Z 54.000,A 180.000,B 0.000,C 180.000} C_DIS
LIN {X 152.480,Y 75.802,Z 54.000,A 180.000,B 0.000,C 180.000} C_DIS
LIN {X 152.475,Y 75.623,Z 54.000,A 180.000,B 0.000,C 180.000} C_DIS
LIN {X 152.419,Y 74.014,Z 54.000,A 180.000,B 0.000,C 180.000} C_DIS
LIN {X 152.409,Y 73.835,Z 54.000,A 180.000,B 0.000,C 180.000} C_DIS
LIN {X 152.325,Y 72.405,Z 54.000,A 180.000,B 0.000,C 180.000} C_DIS
LIN {X 152.315,Y 72.239,Z 54.000,A 180.000,B 0.000,C 180.000} C_DIS
LIN {X 152.314,Y 72.226,Z 54.000,A 180.000,B 0.000,C 180.000} C_DIS
LIN {X 152.300,Y 72.048,Z 54.000,A 180.000,B 0.000,C 180.000} C_DIS
LIN {X 152.182,Y 70.617,Z 54.000,A 180.000,B 0.000,C 180.000} C_DIS
LIN {X 152.167,Y 70.439,Z 54.000,A 180.000,B 0.000,C 180.000} C_DIS
LIN {X 151.996,Y 68.830,Z 54.000,A 180.000,B 0.000,C 180.000} C_DIS
LIN {X 151.975,Y 68.651,Z 54.000,A 180.000,B 0.000,C 180.000} C_DIS
LIN {X 151.767,Y 67.042,Z 54.000,A 180.000,B 0.000,C 180.000} C_DIS
LIN {X 151.741,Y 66.863,Z 54.000,A 180.000,B 0.000,C 180.000} C_DIS
LIN {X 151.521,Y 65.433,Z 54.000,A 180.000,B 0.000,C 180.000} C_DIS
LIN {X 151.494,Y 65.254,Z 54.000,A 180.000,B 0.000,C 180.000} C_DIS
LIN {X 151.462,Y 65.075,Z 54.000,A 180.000,B 0.000,C 180.000} C_DIS
LIN {X 151.208,Y 63.645,Z 54.000,A 180.000,B 0.000,C 180.000} C_DIS
LIN {X 151.175,Y 63.467,Z 54.000,A 180.000,B 0.000,C 180.000} C_DIS
LIN {X 150.850,Y 61.858,Z 54.000,A 180.000,B 0.000,C 180.000} C_DIS
LIN {X 150.811,Y 61.679,Z 54.000,A 180.000,B 0.000,C 180.000} C_DIS
LIN {X 150.487,Y 60.249,Z 54.000,A 180.000,B 0.000,C 180.000} C_DIS
LIN {X 150.447,Y 60.070,Z 54.000,A 180.000,B 0.000,C 180.000} C_DIS
LIN {X 150.402,Y 59.891,Z 54.000,A 180.000,B 0.000,C 180.000} C_DIS
LIN {X 150.042,Y 58.461,Z 54.000,A 180.000,B 0.000,C 180.000} C_DIS
LIN {X 149.995,Y 58.282,Z 54.000,A 180.000,B 0.000,C 180.000} C_DIS
LIN {X 149.600,Y 56.852,Z 54.000,A 180.000,B 0.000,C 180.000} C_DIS
LIN {X 149.550,Y 56.673,Z 54.000,A 180.000,B 0.000,C 180.000} C_DIS
LIN {X 149.497,Y 56.495,Z 54.000,A 180.000,B 0.000,C 180.000} C_DIS
LIN {X 149.065,Y 55.064,Z 54.000,A 180.000,B 0.000,C 180.000} C_DIS
LIN {X 149.008,Y 54.886,Z 54.000,A 180.000,B 0.000,C 180.000} C_DIS
LIN {X 148.540,Y 53.455,Z 54.000,A 180.000,B 0.000,C 180.000} C_DIS
LIN {X 148.480,Y 53.277,Z 54.000,A 180.000,B 0.000,C 180.000} C_DIS
LIN {X 147.974,Y 51.847,Z 54.000,A 180.000,B 0.000,C 180.000} C_DIS
LIN {X 147.911,Y 51.668,Z 54.000,A 180.000,B 0.000,C 180.000} C_DIS
LIN {X 147.846,Y 51.496,Z 54.000,A 180.000,B 0.000,C 180.000} C_DIS
LIN {X 147.299,Y 50.059,Z 54.000,A 180.000,B 0.000,C 180.000} C_DIS
LIN {X 147.227,Y 49.880,Z 54.000,A 180.000,B 0.000,C 180.000} C_DIS
LIN {X 146.645,Y 48.450,Z 54.000,A 180.000,B 0.000,C 180.000} C_DIS
LIN {X 146.595,Y 48.331,Z 54.000,A 180.000,B 0.000,C 180.000} C_DIS
LIN {X 145.947,Y 46.841,Z 54.000,A 180.000,B 0.000,C 180.000} C_DIS
LIN {X 145.880,Y 46.692,Z 54.000,A 180.000,B 0.000,C 180.000} C_DIS
LIN {X 145.203,Y 45.232,Z 54.000,A 180.000,B 0.000,C 180.000} C_DIS
LIN {X 145.164,Y 45.151,Z 54.000,A 180.000,B 0.000,C 180.000} C_DIS
LIN {X 144.449,Y 43.697,Z 54.000,A 180.000,B 0.000,C 180.000} C_DIS
LIN {X 144.413,Y 43.623,Z 54.000,A 180.000,B 0.000,C 180.000} C_DIS
LIN {X 144.320,Y 43.444,Z 54.000,A 180.000,B 0.000,C 180.000} C_DIS
LIN {X 143.668,Y 42.193,Z 54.000,A 180.000,B 0.000,C 180.000} C_DIS
LIN {X 143.574,Y 42.014,Z 54.000,A 180.000,B 0.000,C 180.000} C_DIS
LIN {X 142.785,Y 40.584,Z 54.000,A 180.000,B 0.000,C 180.000} C_DIS
LIN {X 142.683,Y 40.405,Z 54.000,A 180.000,B 0.000,C 180.000} C_DIS
LIN {X 141.947,Y 39.141,Z 54.000,A 180.000,B 0.000,C 180.000} C_DIS
LIN {X 141.849,Y 38.975,Z 54.000,A 180.000,B 0.000,C 180.000} C_DIS
LIN {X 141.768,Y 38.842,Z 54.000,A 180.000,B 0.000,C 180.000} C_DIS
LIN {X 140.971,Y 37.545,Z 54.000,A 180.000,B 0.000,C 180.000} C_DIS
LIN {X 140.874,Y 37.393,Z 54.000,A 180.000,B 0.000,C 180.000} C_DIS
LIN {X 140.047,Y 36.115,Z 54.000,A 180.000,B 0.000,C 180.000} C_DIS
LIN {X 139.980,Y 36.012,Z 54.000,A 180.000,B 0.000,C 180.000} C_DIS
LIN {X 139.928,Y 35.936,Z 54.000,A 180.000,B 0.000,C 180.000} C_DIS
LIN {X 139.076,Y 34.685,Z 54.000,A 180.000,B 0.000,C 180.000} C_DIS
LIN {X 138.953,Y 34.506,Z 54.000,A 180.000,B 0.000,C 180.000} C_DIS
LIN {X 138.014,Y 33.194,Z 54.000,A 180.000,B 0.000,C 180.000} C_DIS
LIN {X 137.927,Y 33.076,Z 54.000,A 180.000,B 0.000,C 180.000} C_DIS
LIN {X 136.941,Y 31.765,Z 54.000,A 180.000,B 0.000,C 180.000} C_DIS
LIN {X 136.848,Y 31.646,Z 54.000,A 180.000,B 0.000,C 180.000} C_DIS
LIN {X 135.861,Y 30.394,Z 54.000,A 180.000,B 0.000,C 180.000} C_DIS
LIN {X 135.714,Y 30.215,Z 54.000,A 180.000,B 0.000,C 180.000} C_DIS
LIN {X 134.796,Y 29.106,Z 54.000,A 180.000,B 0.000,C 180.000} C_DIS
LIN {X 134.677,Y 28.964,Z 54.000,A 180.000,B 0.000,C 180.000} C_DIS
LIN {X 133.590,Y 27.713,Z 54.000,A 180.000,B 0.000,C 180.000} C_DIS
LIN {X 133.544,Y 27.660,Z 54.000,A 180.000,B 0.000,C 180.000} C_DIS
LIN {X 133.430,Y 27.534,Z 54.000,A 180.000,B 0.000,C 180.000} C_DIS
LIN {X 132.453,Y 26.461,Z 54.000,A 180.000,B 0.000,C 180.000} C_DIS
LIN {X 132.293,Y 26.289,Z 54.000,A 180.000,B 0.000,C 180.000} C_DIS
LIN {X 131.220,Y 25.165,Z 54.000,A 180.000,B 0.000,C 180.000} C_DIS
LIN {X 131.090,Y 25.031,Z 54.000,A 180.000,B 0.000,C 180.000} C_DIS
LIN {X 129.969,Y 23.910,Z 54.000,A 180.000,B 0.000,C 180.000} C_DIS
LIN {X 129.835,Y 23.780,Z 54.000,A 180.000,B 0.000,C 180.000} C_DIS
LIN {X 128.711,Y 22.707,Z 54.000,A 180.000,B 0.000,C 180.000} C_DIS
LIN {X 128.539,Y 22.547,Z 54.000,A 180.000,B 0.000,C 180.000} C_DIS
LIN {X 127.466,Y 21.570,Z 54.000,A 180.000,B 0.000,C 180.000} C_DIS
LIN {X 127.340,Y 21.456,Z 54.000,A 180.000,B 0.000,C 180.000} C_DIS
LIN {X 127.287,Y 21.410,Z 54.000,A 180.000,B 0.000,C 180.000} C_DIS
LIN {X 126.036,Y 20.323,Z 54.000,A 180.000,B 0.000,C 180.000} C_DIS
LIN {X 125.894,Y 20.204,Z 54.000,A 180.000,B 0.000,C 180.000} C_DIS
LIN {X 124.785,Y 19.286,Z 54.000,A 180.000,B 0.000,C 180.000} C_DIS
LIN {X 124.606,Y 19.139,Z 54.000,A 180.000,B 0.000,C 180.000} C_DIS
LIN {X 123.354,Y 18.152,Z 54.000,A 180.000,B 0.000,C 180.000} C_DIS
LIN {X 123.235,Y 18.059,Z 54.000,A 180.000,B 0.000,C 180.000} C_DIS
LIN {X 121.924,Y 17.073,Z 54.000,A 180.000,B 0.000,C 180.000} C_DIS
LIN {X 121.806,Y 16.986,Z 54.000,A 180.000,B 0.000,C 180.000} C_DIS
LIN {X 120.494,Y 16.047,Z 54.000,A 180.000,B 0.000,C 180.000} C_DIS
LIN {X 120.315,Y 15.924,Z 54.000,A 180.000,B 0.000,C 180.000} C_DIS
LIN {X 119.064,Y 15.072,Z 54.000,A 180.000,B 0.000,C 180.000} C_DIS
LIN {X 118.988,Y 15.020,Z 54.000,A 180.000,B 0.000,C 180.000} C_DIS
LIN {X 118.885,Y 14.953,Z 54.000,A 180.000,B 0.000,C 180.000} C_DIS
LIN {X 117.607,Y 14.126,Z 54.000,A 180.000,B 0.000,C 180.000} C_DIS
LIN {X 117.455,Y 14.029,Z 54.000,A 180.000,B 0.000,C 180.000} C_DIS
LIN {X 116.158,Y 13.232,Z 54.000,A 180.000,B 0.000,C 180.000} C_DIS
LIN {X 116.025,Y 13.151,Z 54.000,A 180.000,B 0.000,C 180.000} C_DIS
LIN {X 115.859,Y 13.053,Z 54.000,A 180.000,B 0.000,C 180.000} C_DIS
LIN {X 114.595,Y 12.317,Z 54.000,A 180.000,B 0.000,C 180.000} C_DIS
LIN {X 114.416,Y 12.215,Z 54.000,A 180.000,B 0.000,C 180.000} C_DIS
LIN {X 112.986,Y 11.426,Z 54.000,A 180.000,B 0.000,C 180.000} C_DIS
LIN {X 112.807,Y 11.332,Z 54.000,A 180.000,B 0.000,C 180.000} C_DIS
LIN {X 111.556,Y 10.680,Z 54.000,A 180.000,B 0.000,C 180.000} C_DIS
LIN {X 111.377,Y 10.587,Z 54.000,A 180.000,B 0.000,C 180.000} C_DIS
LIN {X 111.303,Y 10.551,Z 54.000,A 180.000,B 0.000,C 180.000} C_DIS
LIN {X 109.849,Y 9.836,Z 54.000,A 180.000,B 0.000,C 180.000} C_DIS
LIN {X 109.768,Y 9.797,Z 54.000,A 180.000,B 0.000,C 180.000} C_DIS
LIN {X 108.308,Y 9.120,Z 54.000,A 180.000,B 0.000,C 180.000} C_DIS
LIN {X 108.159,Y 9.053,Z 54.000,A 180.000,B 0.000,C 180.000} C_DIS
LIN {X 106.669,Y 8.405,Z 54.000,A 180.000,B 0.000,C 180.000} C_DIS
LIN {X 106.550,Y 8.355,Z 54.000,A 180.000,B 0.000,C 180.000} C_DIS
LIN {X 105.120,Y 7.773,Z 54.000,A 180.000,B 0.000,C 180.000} C_DIS
LIN {X 104.941,Y 7.701,Z 54.000,A 180.000,B 0.000,C 180.000} C_DIS
LIN {X 103.504,Y 7.154,Z 54.000,A 180.000,B 0.000,C 180.000} C_DIS
LIN {X 103.332,Y 7.089,Z 54.000,A 180.000,B 0.000,C 180.000} C_DIS
LIN {X 103.153,Y 7.026,Z 54.000,A 180.000,B 0.000,C 180.000} C_DIS
LIN {X 101.723,Y 6.520,Z 54.000,A 180.000,B 0.000,C 180.000} C_DIS
LIN {X 101.545,Y 6.460,Z 54.000,A 180.000,B 0.000,C 180.000} C_DIS
LIN {X 100.114,Y 5.992,Z 54.000,A 180.000,B 0.000,C 180.000} C_DIS
LIN {X 99.936,Y 5.935,Z 54.000,A 180.000,B 0.000,C 180.000} C_DIS
LIN {X 98.505,Y 5.503,Z 54.000,A 180.000,B 0.000,C 180.000} C_DIS
LIN {X 98.327,Y 5.450,Z 54.000,A 180.000,B 0.000,C 180.000} C_DIS
LIN {X 98.148,Y 5.400,Z 54.000,A 180.000,B 0.000,C 180.000} C_DIS
LIN {X 96.718,Y 5.005,Z 54.000,A 180.000,B 0.000,C 180.000} C_DIS
LIN {X 96.539,Y 4.958,Z 54.000,A 180.000,B 0.000,C 180.000} C_DIS
LIN {X 95.109,Y 4.598,Z 54.000,A 180.000,B 0.000,C 180.000} C_DIS
LIN {X 94.930,Y 4.554,Z 54.000,A 180.000,B 0.000,C 180.000} C_DIS
LIN {X 94.751,Y 4.513,Z 54.000,A 180.000,B 0.000,C 180.000} C_DIS
LIN {X 93.321,Y 4.189,Z 54.000,A 180.000,B 0.000,C 180.000} C_DIS
LIN {X 93.142,Y 4.150,Z 54.000,A 180.000,B 0.000,C 180.000} C_DIS
LIN {X 91.533,Y 3.825,Z 54.000,A 180.000,B 0.000,C 180.000} C_DIS
LIN {X 91.355,Y 3.792,Z 54.000,A 180.000,B 0.000,C 180.000} C_DIS
LIN {X 89.925,Y 3.538,Z 54.000,A 180.000,B 0.000,C 180.000} C_DIS
LIN {X 89.746,Y 3.506,Z 54.000,A 180.000,B 0.000,C 180.000} C_DIS
LIN {X 89.567,Y 3.479,Z 54.000,A 180.000,B 0.000,C 180.000} C_DIS
LIN {X 88.137,Y 3.259,Z 54.000,A 180.000,B 0.000,C 180.000} C_DIS
LIN {X 87.958,Y 3.233,Z 54.000,A 180.000,B 0.000,C 180.000} C_DIS
LIN {X 86.349,Y 3.025,Z 54.000,A 180.000,B 0.000,C 180.000} C_DIS
LIN {X 86.170,Y 3.004,Z 54.000,A 180.000,B 0.000,C 180.000} C_DIS
LIN {X 84.561,Y 2.833,Z 54.000,A 180.000,B 0.000,C 180.000} C_DIS
LIN {X 84.383,Y 2.818,Z 54.000,A 180.000,B 0.000,C 180.000} C_DIS
LIN {X 82.952,Y 2.700,Z 54.000,A 180.000,B 0.000,C 180.000} C_DIS
LIN {X 82.774,Y 2.686,Z 54.000,A 180.000,B 0.000,C 180.000} C_DIS
LIN {X 82.761,Y 2.685,Z 54.000,A 180.000,B 0.000,C 180.000} C_DIS
LIN {X 82.595,Y 2.675,Z 54.000,A 180.000,B 0.000,C 180.000} C_DIS
LIN {X 81.165,Y 2.591,Z 54.000,A 180.000,B 0.000,C 180.000} C_DIS
LIN {X 80.986,Y 2.581,Z 54.000,A 180.000,B 0.000,C 180.000} C_DIS
LIN {X 79.377,Y 2.525,Z 54.000,A 180.000,B 0.000,C 180.000} C_DIS
LIN {X 79.198,Y 2.520,Z 54.000,A 180.000,B 0.000,C 180.000} C_DIS
LIN {X 77.589,Y 2.501,Z 54.000,A 180.000,B 0.000,C 180.000} C_DIS
LIN {X 77.411,Y 2.501,Z 54.000,A 180.000,B 0.000,C 180.000} C_DIS
LIN {X 75.802,Y 2.520,Z 54.000,A 180.000,B 0.000,C 180.000} C_DIS
LIN {X 75.623,Y 2.525,Z 54.000,A 180.000,B 0.000,C 180.000} C_DIS
LIN {X 74.014,Y 2.581,Z 54.000,A 180.000,B 0.000,C 180.000} C_DIS
LIN {X 73.835,Y 2.591,Z 54.000,A 180.000,B 0.000,C 180.000} C_DIS
LIN {X 72.405,Y 2.675,Z 54.000,A 180.000,B 0.000,C 180.000} C_DIS
LIN {X 72.239,Y 2.685,Z 54.000,A 180.000,B 0.000,C 180.000} C_DIS
LIN {X 72.226,Y 2.686,Z 54.000,A 180.000,B 0.000,C 180.000} C_DIS
LIN {X 72.048,Y 2.700,Z 54.000,A 180.000,B 0.000,C 180.000} C_DIS
LIN {X 70.617,Y 2.818,Z 54.000,A 180.000,B 0.000,C 180.000} C_DIS
LIN {X 70.439,Y 2.833,Z 54.000,A 180.000,B 0.000,C 180.000} C_DIS
LIN {X 68.830,Y 3.004,Z 54.000,A 180.000,B 0.000,C 180.000} C_DIS
LIN {X 68.651,Y 3.025,Z 54.000,A 180.000,B 0.000,C 180.000} C_DIS
LIN {X 67.042,Y 3.233,Z 54.000,A 180.000,B 0.000,C 180.000} C_DIS
LIN {X 66.863,Y 3.259,Z 54.000,A 180.000,B 0.000,C 180.000} C_DIS
LIN {X 65.433,Y 3.479,Z 54.000,A 180.000,B 0.000,C 180.000} C_DIS
LIN {X 65.254,Y 3.506,Z 54.000,A 180.000,B 0.000,C 180.000} C_DIS
LIN {X 65.075,Y 3.538,Z 54.000,A 180.000,B 0.000,C 180.000} C_DIS
LIN {X 63.645,Y 3.792,Z 54.000,A 180.000,B 0.000,C 180.000} C_DIS
LIN {X 63.467,Y 3.825,Z 54.000,A 180.000,B 0.000,C 180.000} C_DIS
LIN {X 61.858,Y 4.150,Z 54.000,A 180.000,B 0.000,C 180.000} C_DIS
LIN {X 61.679,Y 4.189,Z 54.000,A 180.000,B 0.000,C 180.000} C_DIS
LIN {X 60.249,Y 4.513,Z 54.000,A 180.000,B 0.000,C 180.000} C_DIS
LIN {X 60.070,Y 4.554,Z 54.000,A 180.000,B 0.000,C 180.000} C_DIS
LIN {X 59.891,Y 4.598,Z 54.000,A 180.000,B 0.000,C 180.000} C_DIS
LIN {X 58.461,Y 4.958,Z 54.000,A 180.000,B 0.000,C 180.000} C_DIS
LIN {X 58.282,Y 5.005,Z 54.000,A 180.000,B 0.000,C 180.000} C_DIS
LIN {X 56.852,Y 5.400,Z 54.000,A 180.000,B 0.000,C 180.000} C_DIS
LIN {X 56.673,Y 5.450,Z 54.000,A 180.000,B 0.000,C 180.000} C_DIS
LIN {X 56.495,Y 5.503,Z 54.000,A 180.000,B 0.000,C 180.000} C_DIS
LIN {X 55.064,Y 5.935,Z 54.000,A 180.000,B 0.000,C 180.000} C_DIS
LIN {X 54.886,Y 5.992,Z 54.000,A 180.000,B 0.000,C 180.000} C_DIS
LIN {X 53.455,Y 6.460,Z 54.000,A 180.000,B 0.000,C 180.000} C_DIS
LIN {X 53.277,Y 6.520,Z 54.000,A 180.000,B 0.000,C 180.000} C_DIS
LIN {X 51.847,Y 7.026,Z 54.000,A 180.000,B 0.000,C 180.000} C_DIS
LIN {X 51.668,Y 7.089,Z 54.000,A 180.000,B 0.000,C 180.000} C_DIS
LIN {X 51.496,Y 7.154,Z 54.000,A 180.000,B 0.000,C 180.000} C_DIS
LIN {X 50.059,Y 7.701,Z 54.000,A 180.000,B 0.000,C 180.000} C_DIS
LIN {X 49.880,Y 7.773,Z 54.000,A 180.000,B 0.000,C 180.000} C_DIS
LIN {X 48.450,Y 8.355,Z 54.000,A 180.000,B 0.000,C 180.000} C_DIS
LIN {X 48.331,Y 8.405,Z 54.000,A 180.000,B 0.000,C 180.000} C_DIS
LIN {X 46.841,Y 9.053,Z 54.000,A 180.000,B 0.000,C 180.000} C_DIS
LIN {X 46.692,Y 9.120,Z 54.000,A 180.000,B 0.000,C 180.000} C_DIS
LIN {X 45.232,Y 9.797,Z 54.000,A 180.000,B 0.000,C 180.000} C_DIS
LIN {X 45.151,Y 9.836,Z 54.000,A 180.000,B 0.000,C 180.000} C_DIS
LIN {X 43.697,Y 10.551,Z 54.000,A 180.000,B 0.000,C 180.000} C_DIS
LIN {X 43.623,Y 10.587,Z 54.000,A 180.000,B 0.000,C 180.000} C_DIS
LIN {X 43.444,Y 10.680,Z 54.000,A 180.000,B 0.000,C 180.000} C_DIS
LIN {X 42.193,Y 11.332,Z 54.000,A 180.000,B 0.000,C 180.000} C_DIS
LIN {X 42.014,Y 11.426,Z 54.000,A 180.000,B 0.000,C 180.000} C_DIS
LIN {X 40.584,Y 12.215,Z 54.000,A 180.000,B 0.000,C 180.000} C_DIS
LIN {X 40.405,Y 12.317,Z 54.000,A 180.000,B 0.000,C 180.000} C_DIS
LIN {X 39.141,Y 13.053,Z 54.000,A 180.000,B 0.000,C 180.000} C_DIS
LIN {X 38.975,Y 13.151,Z 54.000,A 180.000,B 0.000,C 180.000} C_DIS
LIN {X 38.842,Y 13.232,Z 54.000,A 180.000,B 0.000,C 180.000} C_DIS
LIN {X 37.545,Y 14.029,Z 54.000,A 180.000,B 0.000,C 180.000} C_DIS
LIN {X 37.393,Y 14.126,Z 54.000,A 180.000,B 0.000,C 180.000} C_DIS
LIN {X 36.115,Y 14.953,Z 54.000,A 180.000,B 0.000,C 180.000} C_DIS
LIN {X 36.012,Y 15.020,Z 54.000,A 180.000,B 0.000,C 180.000} C_DIS
LIN {X 35.936,Y 15.072,Z 54.000,A 180.000,B 0.000,C 180.000} C_DIS
LIN {X 34.685,Y 15.924,Z 54.000,A 180.000,B 0.000,C 180.000} C_DIS
LIN {X 34.506,Y 16.047,Z 54.000,A 180.000,B 0.000,C 180.000} C_DIS
LIN {X 33.194,Y 16.986,Z 54.000,A 180.000,B 0.000,C 180.000} C_DIS
LIN {X 33.076,Y 17.073,Z 54.000,A 180.000,B 0.000,C 180.000} C_DIS
LIN {X 31.765,Y 18.059,Z 54.000,A 180.000,B 0.000,C 180.000} C_DIS
LIN {X 31.646,Y 18.152,Z 54.000,A 180.000,B 0.000,C 180.000} C_DIS
LIN {X 30.394,Y 19.139,Z 54.000,A 180.000,B 0.000,C 180.000} C_DIS
LIN {X 30.215,Y 19.286,Z 54.000,A 180.000,B 0.000,C 180.000} C_DIS
LIN {X 29.106,Y 20.204,Z 54.000,A 180.000,B 0.000,C 180.000} C_DIS
LIN {X 28.964,Y 20.323,Z 54.000,A 180.000,B 0.000,C 180.000} C_DIS
LIN {X 27.713,Y 21.410,Z 54.000,A 180.000,B 0.000,C 180.000} C_DIS
LIN {X 27.660,Y 21.456,Z 54.000,A 180.000,B 0.000,C 180.000} C_DIS
LIN {X 27.534,Y 21.570,Z 54.000,A 180.000,B 0.000,C 180.000} C_DIS
LIN {X 26.461,Y 22.547,Z 54.000,A 180.000,B 0.000,C 180.000} C_DIS
LIN {X 26.289,Y 22.707,Z 54.000,A 180.000,B 0.000,C 180.000} C_DIS
LIN {X 25.165,Y 23.780,Z 54.000,A 180.000,B 0.000,C 180.000} C_DIS
LIN {X 25.031,Y 23.910,Z 54.000,A 180.000,B 0.000,C 180.000} C_DIS
LIN {X 23.910,Y 25.031,Z 54.000,A 180.000,B 0.000,C 180.000} C_DIS
LIN {X 23.780,Y 25.165,Z 54.000,A 180.000,B 0.000,C 180.000} C_DIS
LIN {X 22.707,Y 26.289,Z 54.000,A 180.000,B 0.000,C 180.000} C_DIS
LIN {X 22.547,Y 26.461,Z 54.000,A 180.000,B 0.000,C 180.000} C_DIS
LIN {X 21.570,Y 27.534,Z 54.000,A 180.000,B 0.000,C 180.000} C_DIS
LIN {X 21.456,Y 27.660,Z 54.000,A 180.000,B 0.000,C 180.000} C_DIS
LIN {X 21.410,Y 27.713,Z 54.000,A 180.000,B 0.000,C 180.000} C_DIS
LIN {X 20.323,Y 28.964,Z 54.000,A 180.000,B 0.000,C 180.000} C_DIS
LIN {X 20.204,Y 29.106,Z 54.000,A 180.000,B 0.000,C 180.000} C_DIS
LIN {X 19.286,Y 30.215,Z 54.000,A 180.000,B 0.000,C 180.000} C_DIS
LIN {X 19.139,Y 30.394,Z 54.000,A 180.000,B 0.000,C 180.000} C_DIS
LIN {X 18.152,Y 31.646,Z 54.000,A 180.000,B 0.000,C 180.000} C_DIS
LIN {X 18.059,Y 31.765,Z 54.000,A 180.000,B 0.000,C 180.000} C_DIS
LIN {X 17.073,Y 33.076,Z 54.000,A 180.000,B 0.000,C 180.000} C_DIS
LIN {X 16.986,Y 33.194,Z 54.000,A 180.000,B 0.000,C 180.000} C_DIS
LIN {X 16.047,Y 34.506,Z 54.000,A 180.000,B 0.000,C 180.000} C_DIS
LIN {X 15.924,Y 34.685,Z 54.000,A 180.000,B 0.000,C 180.000} C_DIS
LIN {X 15.072,Y 35.936,Z 54.000,A 180.000,B 0.000,C 180.000} C_DIS
LIN {X 15.020,Y 36.012,Z 54.000,A 180.000,B 0.000,C 180.000} C_DIS
LIN {X 14.953,Y 36.115,Z 54.000,A 180.000,B 0.000,C 180.000} C_DIS
LIN {X 14.126,Y 37.393,Z 54.000,A 180.000,B 0.000,C 180.000} C_DIS
LIN {X 14.029,Y 37.545,Z 54.000,A 180.000,B 0.000,C 180.000} C_DIS
LIN {X 13.232,Y 38.842,Z 54.000,A 180.000,B 0.000,C 180.000} C_DIS
LIN {X 13.151,Y 38.975,Z 54.000,A 180.000,B 0.000,C 180.000} C_DIS
LIN {X 13.053,Y 39.141,Z 54.000,A 180.000,B 0.000,C 180.000} C_DIS
LIN {X 12.317,Y 40.405,Z 54.000,A 180.000,B 0.000,C 180.000} C_DIS
LIN {X 12.215,Y 40.584,Z 54.000,A 180.000,B 0.000,C 180.000} C_DIS
LIN {X 11.426,Y 42.014,Z 54.000,A 180.000,B 0.000,C 180.000} C_DIS
LIN {X 11.332,Y 42.193,Z 54.000,A 180.000,B 0.000,C 180.000} C_DIS
LIN {X 10.680,Y 43.444,Z 54.000,A 180.000,B 0.000,C 180.000} C_DIS
LIN {X 10.587,Y 43.623,Z 54.000,A 180.000,B 0.000,C 180.000} C_DIS
LIN {X 10.551,Y 43.697,Z 54.000,A 180.000,B 0.000,C 180.000} C_DIS
LIN {X 9.836,Y 45.151,Z 54.000,A 180.000,B 0.000,C 180.000} C_DIS
LIN {X 9.797,Y 45.232,Z 54.000,A 180.000,B 0.000,C 180.000} C_DIS
LIN {X 9.120,Y 46.692,Z 54.000,A 180.000,B 0.000,C 180.000} C_DIS
LIN {X 9.053,Y 46.841,Z 54.000,A 180.000,B 0.000,C 180.000} C_DIS
LIN {X 8.405,Y 48.331,Z 54.000,A 180.000,B 0.000,C 180.000} C_DIS
LIN {X 8.355,Y 48.450,Z 54.000,A 180.000,B 0.000,C 180.000} C_DIS
LIN {X 7.773,Y 49.880,Z 54.000,A 180.000,B 0.000,C 180.000} C_DIS
LIN {X 7.701,Y 50.059,Z 54.000,A 180.000,B 0.000,C 180.000} C_DIS
LIN {X 7.154,Y 51.496,Z 54.000,A 180.000,B 0.000,C 180.000} C_DIS
LIN {X 7.089,Y 51.668,Z 54.000,A 180.000,B 0.000,C 180.000} C_DIS
LIN {X 7.026,Y 51.847,Z 54.000,A 180.000,B 0.000,C 180.000} C_DIS
LIN {X 6.520,Y 53.277,Z 54.000,A 180.000,B 0.000,C 180.000} C_DIS
LIN {X 6.460,Y 53.455,Z 54.000,A 180.000,B 0.000,C 180.000} C_DIS
LIN {X 5.992,Y 54.886,Z 54.000,A 180.000,B 0.000,C 180.000} C_DIS
LIN {X 5.935,Y 55.064,Z 54.000,A 180.000,B 0.000,C 180.000} C_DIS
LIN {X 5.503,Y 56.495,Z 54.000,A 180.000,B 0.000,C 180.000} C_DIS
LIN {X 5.450,Y 56.673,Z 54.000,A 180.000,B 0.000,C 180.000} C_DIS
LIN {X 5.400,Y 56.852,Z 54.000,A 180.000,B 0.000,C 180.000} C_DIS
LIN {X 5.005,Y 58.282,Z 54.000,A 180.000,B 0.000,C 180.000} C_DIS
LIN {X 4.958,Y 58.461,Z 54.000,A 180.000,B 0.000,C 180.000} C_DIS
LIN {X 4.598,Y 59.891,Z 54.000,A 180.000,B 0.000,C 180.000} C_DIS
LIN {X 4.554,Y 60.070,Z 54.000,A 180.000,B 0.000,C 180.000} C_DIS
LIN {X 4.513,Y 60.249,Z 54.000,A 180.000,B 0.000,C 180.000} C_DIS
LIN {X 4.189,Y 61.679,Z 54.000,A 180.000,B 0.000,C 180.000} C_DIS
LIN {X 4.150,Y 61.858,Z 54.000,A 180.000,B 0.000,C 180.000} C_DIS
LIN {X 3.825,Y 63.467,Z 54.000,A 180.000,B 0.000,C 180.000} C_DIS
LIN {X 3.792,Y 63.645,Z 54.000,A 180.000,B 0.000,C 180.000} C_DIS
LIN {X 3.538,Y 65.075,Z 54.000,A 180.000,B 0.000,C 180.000} C_DIS
LIN {X 3.506,Y 65.254,Z 54.000,A 180.000,B 0.000,C 180.000} C_DIS
LIN {X 3.479,Y 65.433,Z 54.000,A 180.000,B 0.000,C 180.000} C_DIS
LIN {X 3.259,Y 66.863,Z 54.000,A 180.000,B 0.000,C 180.000} C_DIS
LIN {X 3.233,Y 67.042,Z 54.000,A 180.000,B 0.000,C 180.000} C_DIS
LIN {X 3.025,Y 68.651,Z 54.000,A 180.000,B 0.000,C 180.000} C_DIS
LIN {X 3.004,Y 68.830,Z 54.000,A 180.000,B 0.000,C 180.000} C_DIS
LIN {X 2.833,Y 70.439,Z 54.000,A 180.000,B 0.000,C 180.000} C_DIS
LIN {X 2.818,Y 70.617,Z 54.000,A 180.000,B 0.000,C 180.000} C_DIS
LIN {X 2.700,Y 72.048,Z 54.000,A 180.000,B 0.000,C 180.000} C_DIS
LIN {X 2.686,Y 72.226,Z 54.000,A 180.000,B 0.000,C 180.000} C_DIS
LIN {X 2.685,Y 72.239,Z 54.000,A 180.000,B 0.000,C 180.000} C_DIS
LIN {X 2.675,Y 72.405,Z 54.000,A 180.000,B 0.000,C 180.000} C_DIS
LIN {X 2.591,Y 73.835,Z 54.000,A 180.000,B 0.000,C 180.000} C_DIS
LIN {X 2.581,Y 74.014,Z 54.000,A 180.000,B 0.000,C 180.000} C_DIS
LIN {X 2.525,Y 75.623,Z 54.000,A 180.000,B 0.000,C 180.000} C_DIS
LIN {X 2.520,Y 75.802,Z 54.000,A 180.000,B 0.000,C 180.000} C_DIS
LIN {X 2.506,Y 76.973,Z 54.000,A 180.000,B 0.000,C 180.000} C_DIS
LIN {X 2.501,Y 77.411,Z 54.000,A 180.000,B 0.000,C 180.000} C_DIS
LIN {X 2.501,Y 77.589,Z 54.000,A 180.000,B 0.000,C 180.000} C_DIS
LIN {X 2.520,Y 79.198,Z 54.000,A 180.000,B 0.000,C 180.000} C_DIS
